C07277=1066.009,101.637,426.334,172.572,27.825,155.091
C07278=1066.003,101.388,426.354,172.570,27.822,155.091
C07279=1065.997,101.139,426.372,172.568,27.819,155.090
C07280=1065.992,100.890,426.391,172.567,27.816,155.090
C07281=1065.985,100.641,426.410,172.565,27.813,155.090
C07282=1065.979,100.391,426.429,172.564,27.811,155.089
C07283=1065.973,100.142,426.448,172.562,27.808,155.089
C07284=1065.967,99.893,426.467,172.561,27.806,155.088
C07285=1065.962,99.645,426.485,172.559,27.803,155.088
C07286=1065.956,99.394,426.504,172.558,27.800,155.088
C07287=1065.950,99.145,426.522,172.556,27.797,155.087
C07288=1065.944,98.896,426.542,172.555,27.794,155.087
C07289=1065.938,98.647,426.560,172.553,27.792,155.086
C07290=1065.933,98.398,426.579,172.551,27.789,155.086
C07291=1065.926,98.149,426.598,172.550,27.787,155.086
C07292=1065.921,97.899,426.616,172.548,27.784,155.085
C07293=1065.914,97.650,426.635,172.547,27.781,155.085
C07294=1065.909,97.400,426.654,172.545,27.778,155.085
C07295=1065.903,97.152,426.673,172.544,27.775,155.084
C07296=1065.897,96.902,426.692,172.542,27.773,155.084
C07297=1065.891,96.653,426.710,172.541,27.770,155.083
C07298=1065.885,96.404,426.728,172.539,27.767,155.083
C07299=1065.879,96.155,426.747,172.538,27.765,155.083
C07300=1065.873,95.906,426.766,172.536,27.762,155.082
C07301=1065.868,95.656,426.784,172.535,27.759,155.082
C07302=1065.861,95.407,426.803,172.533,27.756,155.081
C07303=1065.856,95.158,426.822,172.531,27.754,155.081
C07304=1065.849,94.874,426.843,172.530,27.751,155.081
C07305=1065.843,94.591,426.864,172.529,27.748,155.080
C07306=1065.836,94.307,426.885,172.526,27.745,155.080
C07307=1065.829,94.023,426.906,172.525,27.741,155.079
C07308=1065.823,93.775,426.925,172.523,27.738,155.079
C07309=1065.817,93.525,426.943,172.522,27.736,155.078
C07310=1065.812,93.275,426.962,172.520,27.733,155.078
C07311=1065.806,93.027,426.981,172.519,27.730,155.078
C07312=1065.800,92.777,426.999,172.517,27.728,155.077
C07313=1065.794,92.528,427.018,172.515,27.725,155.077
C07314=1065.788,92.279,427.036,172.514,27.722,155.077
C07315=1065.783,92.029,427.055,172.512,27.719,155.076
C07316=1065.776,91.780,427.073,172.511,27.717,155.076
C07317=1065.772,91.531,427.091,172.510,27.714,155.075
C07318=1065.765,91.282,427.110,172.509,27.711,155.075
C07319=1065.759,91.033,427.129,172.507,27.708,155.075
C07320=1065.754,90.783,427.147,172.506,27.706,155.074
C07321=1065.748,90.534,427.166,172.504,27.703,155.074
C07322=1065.741,90.284,427.184,172.503,27.700,155.073
C07323=1065.736,90.036,427.202,172.501,27.697,155.073
C07324=1065.730,89.786,427.220,172.499,27.695,155.073
C07325=1065.724,89.537,427.239,172.498,27.692,155.072
C07326=1065.717,89.288,427.258,172.496,27.689,155.072
C07327=1065.712,89.039,427.275,172.495,27.687,155.071
C07328=1065.705,88.790,427.294,172.493,27.684,155.071
C07329=1065.700,88.540,427.312,172.492,27.681,155.071
C07330=1065.694,88.291,427.331,172.490,27.679,155.070
C07331=1065.688,88.041,427.349,172.489,27.676,155.070
C07332=1065.682,87.792,427.367,172.487,27.673,155.070
C07333=1065.676,87.543,427.385,172.486,27.670,155.069
C07334=1065.670,87.293,427.403,172.484,27.668,155.069
C07335=1065.664,87.044,427.422,172.483,27.665,155.068
C07336=1065.659,86.795,427.440,172.481,27.663,155.068
C07337=1065.652,86.546,427.458,172.480,27.660,155.068
C07338=1065.647,86.297,427.476,172.478,27.657,155.067
C07339=1065.640,86.048,427.494,172.476,27.654,155.067
C07340=1065.634,85.798,427.512,172.476,27.652,155.066
C07341=1065.629,85.549,427.530,172.474,27.649,155.066
C07342=1065.623,85.299,427.549,172.473,27.646,155.066
C07343=1065.617,85.050,427.567,172.471,27.643,155.065
C07344=1065.611,84.801,427.585,172.470,27.641,155.065
C07345=1065.605,84.552,427.603,172.468,27.638,155.065
C07346=1065.600,84.303,427.621,172.467,27.635,155.064
C07347=1065.593,84.053,427.640,172.465,27.633,155.064
C07348=1065.588,83.804,427.657,172.464,27.630,155.063
C07349=1065.582,83.554,427.676,172.462,27.627,155.063
C07350=1065.576,83.305,427.694,172.461,27.624,155.063
C07351=1065.570,83.056,427.712,172.459,27.621,155.062
C07352=1065.564,82.806,427.730,172.458,27.619,155.062
C07353=1065.558,82.558,427.748,172.456,27.616,155.062
C07354=1065.552,82.308,427.766,172.454,27.614,155.061
C07355=1065.547,82.059,427.784,172.453,27.611,155.061
C07356=1065.541,81.809,427.801,172.451,27.608,155.060
C07357=1065.535,81.561,427.820,172.451,27.605,155.060
C07358=1065.529,81.311,427.838,172.449,27.603,155.059
C07359=1065.523,81.061,427.856,172.448,27.600,155.059
C07360=1065.517,80.813,427.875,172.446,27.597,155.059
C07361=1065.511,80.563,427.892,172.445,27.594,155.058
C07362=1065.506,80.314,427.910,172.443,27.591,155.058
C07363=1065.500,80.064,427.928,172.442,27.589,155.058
C07364=1065.494,79.815,427.946,172.440,27.586,155.057
C07365=1065.488,79.566,427.964,172.439,27.583,155.057
C07366=1065.482,79.317,427.982,172.437,27.581,155.056
C07367=1065.476,79.067,428.000,172.436,27.578,155.056
C07368=1065.470,78.784,428.020,172.434,27.575,155.056
C07369=1065.464,78.500,428.040,172.433,27.572,155.055
C07370=1065.456,78.217,428.060,172.431,27.568,155.055
C07371=1065.449,77.933,428.081,172.429,27.565,155.054
C07372=1065.444,77.684,428.099,172.427,27.563,155.054
C07373=1065.438,77.435,428.117,172.427,27.560,155.053
C07374=1065.432,77.186,428.134,172.425,27.557,155.053
C07375=1065.426,76.936,428.152,172.424,27.555,155.053
C07376=1065.420,76.687,428.169,172.422,27.552,155.052
C07377=1065.414,76.437,428.187,172.421,27.549,155.052
C07378=1065.408,76.189,428.205,172.419,27.547,155.052
C07379=1065.402,75.939,428.223,172.418,27.544,155.051
C07380=1065.396,75.690,428.241,172.416,27.541,155.051
C07381=1065.390,75.440,428.259,172.415,27.539,155.050
C07382=1065.385,75.191,428.276,172.413,27.536,155.050
C07383=1065.379,74.942,428.294,172.412,27.533,155.050
C07384=1065.372,74.693,428.311,172.410,27.530,155.049
C07385=1065.366,74.443,428.329,172.409,27.527,155.049
C07386=1065.361,74.194,428.347,172.407,27.525,155.048
C07387=1065.355,73.944,428.365,172.406,27.522,155.048
C07388=1065.349,73.695,428.382,172.405,27.520,155.048
C07389=1065.343,73.446,428.400,172.403,27.517,155.047
C07390=1065.337,73.197,428.417,172.402,27.514,155.047
C07391=1065.331,72.948,428.435,172.400,27.511,155.047
C07392=1065.325,72.698,428.453,172.399,27.509,155.046
C07393=1065.320,72.449,428.470,172.397,27.506,155.046
C07394=1065.313,72.199,428.488,172.396,27.503,155.045
C07395=1065.308,71.950,428.506,172.394,27.500,155.045
C07396=1065.301,71.701,428.523,172.393,27.498,155.045
C07397=1065.296,71.452,428.541,172.391,27.495,155.044
C07398=1065.290,71.203,428.558,172.390,27.492,155.044
C07399=1065.284,70.953,428.576,172.388,27.489,155.043
C07400=1065.279,70.703,428.593,172.388,27.487,155.043
C07401=1065.272,70.454,428.610,172.386,27.484,155.043
C07402=1065.266,70.205,428.628,172.385,27.481,155.042
C07403=1065.261,69.956,428.646,172.383,27.479,155.042
C07404=1065.255,69.706,428.664,172.382,27.476,155.042
C07405=1065.248,69.457,428.681,172.380,27.473,155.041
C07406=1065.242,69.208,428.698,172.379,27.471,155.041
C07407=1065.237,68.959,428.716,172.377,27.468,155.040
C07408=1065.230,68.708,428.733,172.376,27.465,155.040
C07409=1065.225,68.459,428.750,172.374,27.463,155.040
C07410=1065.219,68.210,428.768,172.372,27.460,155.039
C07411=1065.212,67.961,428.785,172.371,27.457,155.039
C07412=1065.207,67.712,428.803,172.369,27.454,155.039
C07413=1065.202,67.462,428.820,172.369,27.452,155.038
C07414=1065.195,67.213,428.837,172.367,27.449,155.038
C07415=1065.189,66.964,428.854,172.366,27.447,155.037
C07416=1065.183,66.714,428.872,172.364,27.444,155.037
C07417=1065.177,66.465,428.889,172.363,27.441,155.037
C07418=1065.172,66.216,428.906,172.361,27.438,155.036
C07419=1065.165,65.966,428.924,172.360,27.435,155.036
C07420=1065.159,65.717,428.941,172.358,27.433,155.035
C07421=1065.154,65.468,428.959,172.357,27.430,155.035
C07422=1065.147,65.218,428.975,172.355,27.428,155.035
C07423=1065.142,64.969,428.993,172.354,27.425,155.034
C07424=1065.136,64.720,429.010,172.352,27.422,155.034
C07425=1065.130,64.470,429.027,172.352,27.419,155.034
C07426=1065.124,64.221,429.045,172.350,27.417,155.033
C07427=1065.117,63.972,429.062,172.349,27.414,155.033
C07428=1065.111,63.722,429.078,172.347,27.411,155.032
C07429=1065.106,63.473,429.096,172.346,27.409,155.032
C07430=1065.099,63.224,429.113,172.344,27.406,155.032
C07431=1065.094,62.974,429.130,172.342,27.404,155.031
C07432=1065.087,62.690,429.149,172.341,27.401,155.031
C07433=1065.080,62.407,429.169,172.340,27.397,155.030
C07434=1065.073,62.123,429.188,172.337,27.394,155.030
C07435=1065.066,61.839,429.208,172.336,27.391,155.030
C07436=1065.060,61.590,429.225,172.334,27.389,155.029
C07437=1065.053,61.341,429.242,172.333,27.386,155.029
C07438=1065.047,61.091,429.259,172.332,27.384,155.029
C07439=1065.041,60.843,429.276,172.331,27.381,155.028
C07440=1065.035,60.592,429.292,172.329,27.378,155.028
C07441=1065.029,60.343,429.310,172.327,27.376,155.028
C07442=1065.023,60.095,429.327,172.326,27.373,155.027
C07443=1065.017,59.844,429.344,172.324,27.370,155.027
C07444=1065.011,59.596,429.361,172.323,27.368,155.026
C07445=1065.005,59.346,429.377,172.321,27.365,155.026
C07446=1064.999,59.097,429.395,172.320,27.362,155.026
C07447=1064.993,58.847,429.412,172.318,27.360,155.025
C07448=1064.987,58.598,429.429,172.317,27.357,155.025
C07449=1064.981,58.349,429.445,172.316,27.355,155.025
C07450=1064.974,58.099,429.463,172.315,27.352,155.024
C07451=1064.969,57.850,429.479,172.313,27.349,155.024
C07452=1064.963,57.601,429.497,172.312,27.346,155.023
C07453=1064.957,57.352,429.513,172.310,27.344,155.023
C07454=1064.950,57.102,429.530,172.309,27.341,155.023
C07455=1064.945,56.853,429.547,172.307,27.338,155.022
C07456=1064.939,56.603,429.563,172.306,27.336,155.022
C07457=1064.932,56.354,429.581,172.304,27.333,155.022
C07458=1064.927,56.104,429.597,172.303,27.331,155.021
C07459=1064.921,55.855,429.614,172.301,27.328,155.021
C07460=1064.915,55.606,429.631,172.300,27.325,155.020
C07461=1064.909,55.357,429.648,172.299,27.322,155.020
C07462=1064.903,55.107,429.665,172.298,27.320,155.020
C07463=1064.897,54.858,429.681,172.296,27.317,155.019
C07464=1064.891,54.609,429.699,172.295,27.314,155.019
C07465=1064.885,54.359,429.715,172.293,27.312,155.019
C07466=1064.879,54.109,429.732,172.292,27.309,155.018
C07467=1064.872,53.860,429.749,172.290,27.307,155.018
C07468=1064.867,53.611,429.765,172.288,27.304,155.017
C07469=1064.861,53.361,429.782,172.287,27.301,155.017
C07470=1064.855,53.113,429.799,172.286,27.298,155.017
C07471=1064.849,52.862,429.816,172.285,27.296,155.016
C07472=1064.843,52.613,429.832,172.283,27.293,155.016
C07473=1064.837,52.364,429.849,172.282,27.290,155.016
C07474=1064.831,52.115,429.865,172.280,27.288,155.015
C07475=1064.826,51.865,429.882,172.279,27.285,155.015
C07476=1064.820,51.617,429.899,172.277,27.282,155.015
C07477=1064.813,51.366,429.916,172.276,27.280,155.014
C07478=1064.808,51.117,429.933,172.274,27.277,155.014
C07479=1064.802,50.867,429.949,172.273,27.274,155.013
C07480=1064.796,50.619,429.966,172.271,27.271,155.013
C07481=1064.790,50.369,429.982,172.270,27.269,155.013
C07482=1064.784,50.120,429.999,172.269,27.266,155.012
C07483=1064.779,49.870,430.015,172.268,27.264,155.012
C07484=1064.772,49.621,430.033,172.266,27.261,155.011
C07485=1064.766,49.372,430.049,172.265,27.258,155.011
C07486=1064.760,49.122,430.066,172.263,27.256,155.011
C07487=1064.755,48.873,430.082,172.262,27.253,155.010
C07488=1064.749,48.623,430.098,172.260,27.250,155.010
C07489=1064.742,48.375,430.115,172.259,27.247,155.010
C07490=1064.737,48.125,430.132,172.257,27.244,155.009
C07491=1064.731,47.875,430.148,172.256,27.241,155.009
C07492=1064.725,47.626,430.165,172.255,27.239,155.008
C07493=1064.719,47.377,430.181,172.254,27.237,155.008
C07494=1064.713,47.126,430.198,172.252,27.234,155.008
C07495=1064.707,46.878,430.215,172.251,27.231,155.007
C07496=1064.701,46.594,430.234,172.249,27.228,155.007
C07497=1064.694,46.309,430.252,172.248,27.225,155.006
C07498=1064.687,46.026,430.272,172.245,27.222,155.006
C07499=1064.680,45.742,430.290,172.244,27.219,155.006
C07500=1064.675,45.492,430.306,172.243,27.216,155.005
C07501=1064.669,45.243,430.323,172.241,27.213,155.005
C07502=1064.663,44.994,430.339,172.240,27.210,155.004
C07503=1064.657,44.744,430.355,172.239,27.208,155.004
C07504=1064.651,44.495,430.371,172.237,27.205,155.004
C07505=1064.646,44.245,430.388,172.236,27.203,155.003
C07506=1064.640,43.996,430.405,172.235,27.200,155.003
C07507=1064.634,43.746,430.421,172.233,27.197,155.003
C07508=1064.628,43.497,430.437,172.232,27.194,155.002
C07509=1064.622,43.248,430.453,172.230,27.192,155.002
C07510=1064.616,42.998,430.470,172.228,27.189,155.002
C07511=1064.610,42.749,430.486,172.227,27.186,155.001
C07512=1064.604,42.500,430.502,172.226,27.183,155.001
C07513=1064.598,42.250,430.518,172.225,27.181,155.000
C07514=1064.592,42.001,430.535,172.223,27.179,155.000
C07515=1064.586,41.752,430.551,172.222,27.176,155.000
C07516=1064.580,41.502,430.567,172.220,27.173,154.999
C07517=1064.574,41.253,430.583,172.219,27.171,154.999
C07518=1064.569,41.004,430.600,172.217,27.168,154.999
C07519=1064.563,40.754,430.616,172.216,27.165,154.998
C07520=1064.557,40.505,430.632,172.214,27.163,154.998
C07521=1064.551,40.256,430.648,172.213,27.160,154.998
C07522=1064.545,40.006,430.665,172.211,27.157,154.997
C07523=1064.539,39.757,430.681,172.211,27.154,154.997
C07524=1064.533,39.508,430.697,172.209,27.152,154.996
C07525=1064.527,39.258,430.713,172.208,27.149,154.996
C07526=1064.521,39.008,430.729,172.206,27.146,154.996
C07527=1064.515,38.759,430.745,172.205,27.144,154.995
C07528=1064.509,38.510,430.762,172.203,27.141,154.995
C07529=1064.503,38.260,430.778,172.202,27.139,154.995
C07530=1064.497,38.011,430.794,172.200,27.136,154.994
C07531=1064.491,37.761,430.810,172.199,27.133,154.994
C07532=1064.485,37.512,430.826,172.197,27.131,154.993
C07533=1064.479,37.262,430.841,172.197,27.128,154.993
C07534=1064.473,37.013,430.858,172.195,27.126,154.993
C07535=1064.467,36.764,430.874,172.194,27.123,154.992
C07536=1064.461,36.514,430.890,172.192,27.120,154.992
C07537=1064.455,36.265,430.906,172.191,27.118,154.992
C07538=1064.449,36.015,430.921,172.189,27.115,154.991
C07539=1064.443,35.766,430.938,172.188,27.112,154.991
C07540=1064.437,35.517,430.954,172.186,27.110,154.991
C07541=1064.430,35.268,430.970,172.185,27.107,154.990
C07542=1064.425,35.018,430.985,172.183,27.105,154.990
C07543=1064.419,34.768,431.001,172.182,27.102,154.990
C07544=1064.413,34.519,431.018,172.181,27.099,154.989
C07545=1064.406,34.270,431.033,172.180,27.097,154.989
C07546=1064.400,34.020,431.049,172.178,27.094,154.989
C07547=1064.395,33.771,431.065,172.177,27.091,154.988
C07548=1064.389,33.521,431.081,172.175,27.089,154.988
C07549=1064.382,33.272,431.096,172.174,27.086,154.987
C07550=1064.376,33.022,431.113,172.172,27.083,154.987
C07551=1064.370,32.773,431.129,172.171,27.081,154.987
C07552=1064.365,32.523,431.144,172.169,27.078,154.986
C07553=1064.358,32.274,431.160,172.168,27.075,154.986
C07554=1064.352,32.025,431.176,172.166,27.073,154.986
C07555=1064.346,31.775,431.192,172.166,27.071,154.985
C07556=1064.340,31.525,431.208,172.164,27.068,154.985
C07557=1064.334,31.277,431.223,172.163,27.065,154.985
C07558=1064.329,31.027,431.239,172.161,27.063,154.984
C07559=1064.323,30.778,431.255,172.160,27.060,154.984
C07560=1064.315,30.494,431.273,172.158,27.057,154.983
C07561=1064.309,30.209,431.291,172.157,27.054,154.983
C07562=1064.302,29.925,431.309,172.154,27.051,154.983
C07563=1064.295,29.642,431.327,172.153,27.048,154.982
C07564=1064.290,29.392,431.342,172.151,27.045,154.982
C07565=1064.283,29.143,431.358,172.150,27.042,154.982
C07566=1064.277,28.894,431.374,172.149,27.040,154.981
C07567=1064.271,28.644,431.390,172.148,27.038,154.981
C07568=1064.265,28.395,431.405,172.146,27.035,154.981
C07569=1064.259,28.145,431.421,172.145,27.032,154.980
C07570=1064.254,27.896,431.437,172.143,27.030,154.980
C07571=1064.247,27.646,431.452,172.142,27.027,154.979
C07572=1064.241,27.397,431.468,172.140,27.025,154.979
C07573=1064.235,27.147,431.483,172.139,27.022,154.979
C07574=1064.229,26.898,431.499,172.137,27.019,154.978
C07575=1064.223,26.648,431.514,172.136,27.017,154.978
C07576=1064.217,26.399,431.531,172.134,27.014,154.978
C07577=1064.211,26.149,431.546,172.134,27.012,154.977
C07578=1064.205,25.901,431.561,172.132,27.009,154.977
C07579=1064.199,25.651,431.577,172.131,27.007,154.977
C07580=1064.193,25.401,431.592,172.129,27.004,154.976
C07581=1064.187,25.152,431.608,172.128,27.001,154.976
C07582=1064.181,24.902,431.623,172.126,26.999,154.976
C07583=1064.175,24.653,431.639,172.125,26.996,154.975
C07584=1064.168,24.403,431.654,172.123,26.993,154.975
C07585=1064.163,24.154,431.669,172.122,26.991,154.975
C07586=1064.157,23.905,431.685,172.120,26.988,154.974
C07587=1064.151,23.655,431.701,172.119,26.986,154.974
C07588=1064.144,23.406,431.716,172.118,26.983,154.974
C07589=1064.139,23.156,431.732,172.117,26.981,154.973
C07590=1064.133,22.907,431.746,172.115,26.978,154.973
C07591=1064.127,22.657,431.763,172.114,26.976,154.973
C07592=1064.121,22.408,431.778,172.112,26.973,154.972
C07593=1064.115,22.158,431.793,172.111,26.970,154.972
C07594=1064.108,21.909,431.809,172.109,26.968,154.972
C07595=1064.103,21.659,431.824,172.108,26.965,154.971
C07596=1064.097,21.410,431.839,172.106,26.963,154.971
C07597=1064.090,21.161,431.855,172.105,26.960,154.971
C07598=1064.084,20.911,431.870,172.103,26.957,154.970
C07599=1064.078,20.661,431.885,172.102,26.955,154.970
C07600=1064.073,20.413,431.901,172.101,26.952,154.969
C07601=1064.066,20.163,431.916,172.099,26.950,154.969
C07602=1064.061,19.913,431.931,172.098,26.947,154.969
C07603=1064.054,19.663,431.946,172.096,26.945,154.969
C07604=1064.048,19.415,431.962,172.095,26.942,154.968
C07605=1064.043,19.165,431.977,172.093,26.940,154.968
C07606=1064.036,18.915,431.992,172.092,26.937,154.967
C07607=1064.030,18.666,432.007,172.090,26.935,154.967
C07608=1064.024,18.416,432.023,172.089,26.932,154.967
C07609=1064.018,18.167,432.038,172.087,26.930,154.967
C07610=1064.012,17.917,432.054,172.086,26.927,154.966
C07611=1064.006,17.668,432.068,172.085,26.925,154.966
C07612=1064.000,17.419,432.083,172.084,26.922,154.965
C07613=1063.995,17.169,432.099,172.082,26.920,154.965
C07614=1063.988,16.920,432.114,172.081,26.917,154.965
C07615=1063.982,16.670,432.129,172.079,26.914,154.964
C07616=1063.976,16.421,432.144,172.078,26.912,154.964
C07617=1063.970,16.171,432.159,172.076,26.909,154.964
C07618=1063.964,15.921,432.174,172.075,26.906,154.963
C07619=1063.958,15.672,432.190,172.073,26.904,154.963
C07620=1063.952,15.423,432.205,172.072,26.901,154.963
C07621=1063.946,15.174,432.220,172.070,26.899,154.963
C07622=1063.939,14.924,432.235,172.069,26.896,154.962
C07623=1063.934,14.675,432.250,172.067,26.894,154.962
C07624=1063.927,14.392,432.267,172.066,26.891,154.961
C07625=1063.920,14.110,432.284,172.064,26.888,154.961
C07626=1063.913,13.826,432.302,172.063,26.885,154.961
C07627=1063.907,13.544,432.318,172.061,26.882,154.960
C07628=1063.900,13.295,432.333,172.060,26.880,154.960
C07629=1063.894,13.045,432.348,172.058,26.877,154.960
C07630=1063.887,12.795,432.363,172.057,26.875,154.959
C07631=1063.882,12.546,432.378,172.055,26.873,154.959
C07632=1063.875,12.297,432.393,172.054,26.870,154.959
C07633=1063.869,12.047,432.408,172.052,26.868,154.958
C07634=1063.863,11.798,432.422,172.051,26.865,154.958
C07635=1063.857,11.548,432.438,172.049,26.862,154.958
C07636=1063.851,11.298,432.453,172.048,26.860,154.957
C07637=1063.845,11.049,432.468,172.047,26.858,154.957
C07638=1063.839,10.800,432.482,172.046,26.855,154.957
C07639=1063.833,10.550,432.497,172.044,26.853,154.957
C07640=1063.826,10.301,432.512,172.043,26.850,154.956
C07641=1063.820,10.052,432.527,172.041,26.848,154.956
C07642=1063.814,9.802,432.542,172.040,26.846,154.956
C07643=1063.808,9.552,432.556,172.038,26.843,154.955
C07644=1063.802,9.303,432.570,172.037,26.840,154.955
C07645=1063.796,9.053,432.585,172.035,26.838,154.955
C07646=1063.789,8.803,432.600,172.034,26.835,154.954
C07647=1063.784,8.554,432.615,172.032,26.833,154.954
C07648=1063.778,8.304,432.630,172.031,26.830,154.954
C07649=1063.772,8.055,432.645,172.029,26.828,154.953
C07650=1063.766,7.806,432.660,172.028,26.826,154.953
C07651=1063.759,7.556,432.675,172.026,26.823,154.953
C07652=1063.754,7.307,432.689,172.025,26.821,154.952
C07653=1063.748,7.057,432.704,172.024,26.818,154.952
C07654=1063.741,6.807,432.719,172.022,26.816,154.952
C07655=1063.735,6.558,432.733,172.021,26.813,154.951
C07656=1063.729,6.309,432.748,172.019,26.810,154.951
C07657=1063.723,6.060,432.763,172.018,26.808,154.951
C07658=1063.717,5.810,432.778,172.016,26.806,154.951
C07659=1063.711,5.560,432.792,172.015,26.803,154.950
C07660=1063.705,5.311,432.807,172.013,26.801,154.950
C07661=1063.699,5.061,432.821,172.012,26.798,154.950
C07662=1063.693,4.812,432.836,172.010,26.795,154.949
C07663=1063.686,4.563,432.851,172.009,26.793,154.949
C07664=1063.681,4.313,432.865,172.007,26.790,154.949
C07665=1063.675,4.063,432.880,172.006,26.788,154.948
C07666=1063.668,3.814,432.895,172.005,26.786,154.948
C07667=1063.662,3.565,432.909,172.004,26.783,154.948
C07668=1063.656,3.314,432.924,172.002,26.781,154.947
C07669=1063.650,3.066,432.938,172.001,26.779,154.947
C07670=1063.644,2.816,432.953,171.999,26.776,154.947
C07671=1063.639,2.566,432.967,171.998,26.773,154.946
C07672=1063.632,2.317,432.982,171.996,26.771,154.946
C07673=1063.626,2.068,432.996,171.995,26.768,154.946
C07674=1063.620,1.818,433.011,171.993,26.766,154.945
C07675=1063.615,1.568,433.025,171.992,26.763,154.945
C07676=1063.608,1.319,433.040,171.990,26.761,154.945
C07677=1063.602,1.070,433.055,171.989,26.759,154.945
C07678=1063.596,0.820,433.069,171.987,26.756,154.944
C07679=1063.591,0.571,433.084,171.986,26.753,154.944
C07680=1063.584,0.321,433.099,171.984,26.751,154.944
C07681=1063.579,0.071,433.112,171.983,26.748,154.943
C07682=1063.572,-0.178,433.127,171.982,26.746,154.943
C07683=1063.567,-0.428,433.141,171.981,26.744,154.943
C07684=1063.560,-0.678,433.156,171.979,26.741,154.942
C07685=1063.555,-0.926,433.171,171.978,26.739,154.942
C07686=1063.549,-1.177,433.185,171.976,26.736,154.942
C07687=1063.543,-1.426,433.200,171.975,26.734,154.941
C07688=1063.537,-1.707,433.216,171.973,26.731,154.941
C07689=1063.529,-1.988,433.232,171.971,26.728,154.941
C07690=1063.523,-2.267,433.248,171.969,26.725,154.940
C07691=1063.516,-2.548,433.264,171.968,26.722,154.940
C07692=1063.510,-2.797,433.279,171.966,26.720,154.940
C07693=1063.504,-3.048,433.293,171.965,26.718,154.939
C07694=1063.498,-3.297,433.308,171.963,26.715,154.939
C07695=1063.492,-3.547,433.322,171.962,26.713,154.939
C07696=1063.486,-3.796,433.336,171.960,26.710,154.938
C07697=1063.480,-4.046,433.350,171.959,26.708,154.938
C07698=1063.474,-4.295,433.365,171.957,26.706,154.938
C07699=1063.468,-4.545,433.379,171.957,26.703,154.937
C07700=1063.462,-4.794,433.393,171.955,26.701,154.937
C07701=1063.455,-5.044,433.407,171.954,26.699,154.937
C07702=1063.449,-5.293,433.422,171.952,26.696,154.937
C07703=1063.443,-5.543,433.436,171.950,26.694,154.936
C07704=1063.437,-5.793,433.449,171.949,26.692,154.936
C07705=1063.431,-6.042,433.464,171.947,26.689,154.936
C07706=1063.425,-6.292,433.478,171.946,26.686,154.935
C07707=1063.419,-6.540,433.492,171.944,26.684,154.935
C07708=1063.413,-6.791,433.506,171.943,26.682,154.935
C07709=1063.407,-7.040,433.521,171.941,26.680,154.935
C07710=1063.400,-7.290,433.534,171.940,26.677,154.934
C07711=1063.394,-7.539,433.548,171.938,26.674,154.934
C07712=1063.388,-7.789,433.563,171.937,26.672,154.934
C07713=1063.382,-8.038,433.576,171.935,26.670,154.933
C07714=1063.376,-8.287,433.591,171.934,26.668,154.933
C07715=1063.370,-8.537,433.605,171.932,26.665,154.933
C07716=1063.364,-8.787,433.619,171.931,26.663,154.933
C07717=1063.357,-9.036,433.633,171.929,26.660,154.932
C07718=1063.352,-9.286,433.647,171.928,26.658,154.932
C07719=1063.346,-9.535,433.661,171.926,26.655,154.932
C07720=1063.339,-9.785,433.676,171.925,26.653,154.931
C07721=1063.334,-10.034,433.689,171.924,26.651,154.931
C07722=1063.327,-10.284,433.703,171.922,26.649,154.931
C07723=1063.322,-10.534,433.717,171.921,26.647,154.931
C07724=1063.316,-10.783,433.732,171.919,26.644,154.930
C07725=1063.309,-11.033,433.745,171.918,26.641,154.930
C07726=1063.304,-11.282,433.759,171.916,26.639,154.930
C07727=1063.297,-11.531,433.773,171.915,26.637,154.929
C07728=1063.291,-11.781,433.787,171.913,26.634,154.929
C07729=1063.285,-12.031,433.801,171.912,26.632,154.929
C07730=1063.279,-12.280,433.814,171.910,26.630,154.929
C07731=1063.273,-12.530,433.829,171.909,26.628,154.928
C07732=1063.267,-12.779,433.843,171.907,26.625,154.928
C07733=1063.261,-13.029,433.856,171.906,26.622,154.928
C07734=1063.255,-13.279,433.871,171.904,26.620,154.927
C07735=1063.249,-13.528,433.884,171.903,26.618,154.927
C07736=1063.243,-13.777,433.899,171.901,26.615,154.927
C07737=1063.237,-14.027,433.913,171.900,26.613,154.927
C07738=1063.231,-14.277,433.926,171.898,26.611,154.926
C07739=1063.225,-14.526,433.940,171.896,26.609,154.926
C07740=1063.219,-14.776,433.954,171.895,26.606,154.926
C07741=1063.213,-15.025,433.968,171.894,26.603,154.925
C07742=1063.207,-15.274,433.981,171.892,26.601,154.925
C07743=1063.200,-15.525,433.996,171.890,26.599,154.925
C07744=1063.194,-15.774,434.009,171.889,26.596,154.925
C07745=1063.189,-16.024,434.023,171.887,26.594,154.924
C07746=1063.182,-16.273,434.036,171.886,26.592,154.924
C07747=1063.176,-16.523,434.050,171.884,26.590,154.924
C07748=1063.170,-16.772,434.064,171.883,26.587,154.924
C07749=1063.164,-17.022,434.077,171.882,26.585,154.923
C07750=1063.158,-17.271,434.092,171.881,26.583,154.923
C07751=1063.151,-17.521,434.105,171.879,26.581,154.923
C07752=1063.145,-17.799,434.120,171.877,26.578,154.923
C07753=1063.138,-18.079,434.135,171.875,26.576,154.922
C07754=1063.131,-18.358,434.150,171.874,26.573,154.922
C07755=1063.124,-18.637,434.165,171.872,26.571,154.922
C07756=1063.118,-18.887,434.179,171.871,26.568,154.921
C07757=1063.112,-19.136,434.193,171.869,26.566,154.921
C07758=1063.106,-19.386,434.207,171.868,26.564,154.921
C07759=1063.100,-19.635,434.220,171.866,26.561,154.921
C07760=1063.093,-19.885,434.233,171.864,26.559,154.920
C07761=1063.088,-20.135,434.247,171.863,26.557,154.920
C07762=1063.082,-20.384,434.261,171.861,26.554,154.920
C07763=1063.075,-20.633,434.274,171.860,26.553,154.920
C07764=1063.069,-20.884,434.288,171.858,26.550,154.919
C07765=1063.063,-21.133,434.301,171.857,26.548,154.919
C07766=1063.058,-21.382,434.315,171.855,26.546,154.919
C07767=1063.051,-21.632,434.328,171.854,26.543,154.919
C07768=1063.045,-21.882,434.342,171.852,26.541,154.918
C07769=1063.039,-22.131,434.356,171.851,26.539,154.918
C07770=1063.033,-22.380,434.369,171.849,26.537,154.918
C07771=1063.027,-22.630,434.382,171.848,26.534,154.917
C07772=1063.021,-22.879,434.396,171.846,26.532,154.917
C07773=1063.014,-23.129,434.410,171.844,26.530,154.917
C07774=1063.008,-23.379,434.423,171.843,26.527,154.917
C07775=1063.003,-23.629,434.436,171.841,26.525,154.916
C07776=1062.997,-23.878,434.450,171.840,26.523,154.916
C07777=1062.991,-24.127,434.463,171.838,26.520,154.916
C07778=1062.985,-24.377,434.477,171.837,26.518,154.916
C07779=1062.978,-24.627,434.490,171.835,26.516,154.915
C07780=1062.972,-24.876,434.504,171.834,26.514,154.915
C07781=1062.966,-25.125,434.517,171.832,26.512,154.915
C07782=1062.961,-25.376,434.530,171.831,26.509,154.915
C07783=1062.954,-25.625,434.543,171.829,26.507,154.914
C07784=1062.948,-25.874,434.557,171.827,26.505,154.914
C07785=1062.942,-26.124,434.571,171.826,26.502,154.914
C07786=1062.936,-26.374,434.584,171.824,26.500,154.914
C07787=1062.930,-26.623,434.597,171.823,26.498,154.913
C07788=1062.925,-26.873,434.611,171.821,26.496,154.913
C07789=1062.918,-27.122,434.624,171.820,26.494,154.913
C07790=1062.912,-27.372,434.637,171.818,26.491,154.913
C07791=1062.905,-27.622,434.651,171.817,26.489,154.912
C07792=1062.899,-27.871,434.663,171.815,26.487,154.912
C07793=1062.893,-28.121,434.677,171.814,26.485,154.912
C07794=1062.887,-28.370,434.690,171.812,26.483,154.912
C07795=1062.881,-28.619,434.703,171.810,26.480,154.911
C07796=1062.875,-28.869,434.716,171.809,26.478,154.911
C07797=1062.869,-29.118,434.729,171.807,26.476,154.911
C07798=1062.863,-29.369,434.743,171.806,26.474,154.911
C07799=1062.857,-29.619,434.756,171.804,26.472,154.910
C07800=1062.850,-29.868,434.769,171.803,26.470,154.910
C07801=1062.844,-30.117,434.782,171.801,26.468,154.910
C07802=1062.838,-30.367,434.795,171.800,26.465,154.910
C07803=1062.832,-30.616,434.808,171.798,26.463,154.910
C07804=1062.826,-30.865,434.821,171.796,26.461,154.909
C07805=1062.819,-31.116,434.834,171.795,26.459,154.909
C07806=1062.813,-31.365,434.848,171.793,26.457,154.909
C07807=1062.807,-31.615,434.861,171.792,26.454,154.909
C07808=1062.801,-31.864,434.873,171.790,26.452,154.908
C07809=1062.795,-32.114,434.887,171.789,26.450,154.908
C07810=1062.789,-32.364,434.899,171.787,26.448,154.908
C07811=1062.783,-32.613,434.912,171.786,26.446,154.908
C07812=1062.776,-32.862,434.926,171.784,26.444,154.907
C07813=1062.771,-33.112,434.939,171.782,26.442,154.907
C07814=1062.765,-33.362,434.952,171.781,26.439,154.907
C07815=1062.759,-33.611,434.965,171.779,26.437,154.907
C07816=1062.752,-33.890,434.979,171.778,26.435,154.906
C07817=1062.745,-34.168,434.994,171.776,26.432,154.906
C07818=1062.738,-34.446,435.009,171.775,26.430,154.906
C07819=1062.731,-34.724,435.023,171.773,26.428,154.906
C07820=1062.725,-34.974,435.035,171.772,26.426,154.905
C07821=1062.720,-35.224,435.049,171.770,26.424,154.905
C07822=1062.714,-35.473,435.062,171.769,26.421,154.905
C07823=1062.708,-35.723,435.075,171.767,26.420,154.905
C07824=1062.702,-35.973,435.088,171.765,26.417,154.905
C07825=1062.695,-36.222,435.101,171.763,26.415,154.904
C07826=1062.690,-36.472,435.113,171.761,26.413,154.904
C07827=1062.683,-36.721,435.127,171.760,26.411,154.904
C07828=1062.677,-36.971,435.139,171.758,26.408,154.904
C07829=1062.671,-37.220,435.152,171.757,26.407,154.904
C07830=1062.665,-37.470,435.165,171.755,26.404,154.903
C07831=1062.659,-37.719,435.178,171.754,26.402,154.903
C07832=1062.653,-37.969,435.191,171.752,26.400,154.903
C07833=1062.647,-38.219,435.203,171.750,26.398,154.903
C07834=1062.641,-38.468,435.217,171.749,26.396,154.902
C07835=1062.635,-38.718,435.229,171.747,26.394,154.902
C07836=1062.628,-38.967,435.242,171.746,26.392,154.902
C07837=1062.622,-39.217,435.254,171.744,26.390,154.902
C07838=1062.616,-39.467,435.267,171.743,26.388,154.901
C07839=1062.610,-39.716,435.280,171.741,26.386,154.901
C07840=1062.604,-39.966,435.293,171.739,26.384,154.901
C07841=1062.598,-40.216,435.305,171.738,26.382,154.901
C07842=1062.591,-40.465,435.318,171.736,26.379,154.901
C07843=1062.585,-40.715,435.331,171.735,26.378,154.901
C07844=1062.579,-40.964,435.344,171.733,26.375,154.900
C07845=1062.573,-41.214,435.356,171.731,26.374,154.900
C07846=1062.567,-41.463,435.368,171.730,26.371,154.900
C07847=1062.561,-41.713,435.381,171.728,26.370,154.900
C07848=1062.555,-41.963,435.394,171.727,26.367,154.899
C07849=1062.549,-42.213,435.407,171.725,26.366,154.899
C07850=1062.542,-42.462,435.419,171.724,26.363,154.899
C07851=1062.536,-42.711,435.432,171.722,26.361,154.899
C07852=1062.530,-42.961,435.445,171.720,26.359,154.899
C07853=1062.524,-43.211,435.457,171.719,26.357,154.898
C07854=1062.518,-43.461,435.470,171.717,26.355,154.898
C07855=1062.511,-43.710,435.482,171.716,26.353,154.898
C07856=1062.505,-43.960,435.495,171.714,26.351,154.898
C07857=1062.499,-44.210,435.507,171.713,26.349,154.898
C07858=1062.494,-44.459,435.520,171.711,26.347,154.897
C07859=1062.487,-44.708,435.532,171.709,26.345,154.897
C07860=1062.481,-44.958,435.545,171.708,26.343,154.897
C07861=1062.475,-45.208,435.557,171.706,26.341,154.897
C07862=1062.469,-45.457,435.570,171.705,26.339,154.897
C07863=1062.463,-45.707,435.582,171.703,26.337,154.896
C07864=1062.456,-45.956,435.595,171.701,26.335,154.896
C07865=1062.451,-46.206,435.608,171.700,26.333,154.896
C07866=1062.445,-46.456,435.620,171.698,26.331,154.896
C07867=1062.438,-46.706,435.632,171.697,26.329,154.896
C07868=1062.433,-46.955,435.644,171.695,26.327,154.895
C07869=1062.427,-47.205,435.657,171.694,26.325,154.895
C07870=1062.420,-47.454,435.670,171.692,26.323,154.895
C07871=1062.414,-47.704,435.682,171.690,26.321,154.895
C07872=1062.408,-47.953,435.695,171.689,26.319,154.895
C07873=1062.402,-48.203,435.707,171.687,26.317,154.895
C07874=1062.395,-48.453,435.719,171.686,26.315,154.894
C07875=1062.390,-48.702,435.731,171.684,26.313,154.894
C07876=1062.384,-48.952,435.744,171.682,26.312,154.894
C07877=1062.378,-49.202,435.756,171.681,26.309,154.894
C07878=1062.372,-49.451,435.769,171.679,26.307,154.894
C07879=1062.366,-49.701,435.781,171.678,26.305,154.893
C07880=1062.359,-49.980,435.795,171.675,26.303,154.893
C07881=1062.352,-50.259,435.808,171.674,26.301,154.893
C07882=1062.345,-50.536,435.822,171.672,26.299,154.893
C07883=1062.338,-50.815,435.836,171.671,26.297,154.893
C07884=1062.333,-51.065,435.848,171.669,26.295,154.892
C07885=1062.326,-51.314,435.860,171.666,26.293,154.892
C07886=1062.319,-51.564,435.872,171.665,26.291,154.892
C07887=1062.313,-51.814,435.885,171.663,26.289,154.892
C07888=1062.307,-52.063,435.897,171.662,26.287,154.892
C07889=1062.301,-52.313,435.909,171.660,26.285,154.892
C07890=1062.294,-52.563,435.921,171.658,26.284,154.891
C07891=1062.289,-52.813,435.933,171.657,26.282,154.891
C07892=1062.282,-53.062,435.945,171.655,26.280,154.891
C07893=1062.276,-53.312,435.957,171.653,26.278,154.891
C07894=1062.270,-53.562,435.969,171.652,26.276,154.891
C07895=1062.263,-53.811,435.981,171.650,26.274,154.891
C07896=1062.257,-54.061,435.994,171.649,26.273,154.890
C07897=1062.251,-54.311,436.006,171.647,26.271,154.890
C07898=1062.245,-54.559,436.017,171.645,26.269,154.890
C07899=1062.239,-54.809,436.030,171.644,26.267,154.890
C07900=1062.232,-55.059,436.042,171.642,26.265,154.890
C07901=1062.225,-55.308,436.054,171.641,26.263,154.890
C07902=1062.220,-55.559,436.066,171.639,26.262,154.889
C07903=1062.214,-55.808,436.077,171.637,26.260,154.889
C07904=1062.208,-56.058,436.090,171.636,26.258,154.889
C07905=1062.201,-56.307,436.102,171.634,26.256,154.889
C07906=1062.195,-56.557,436.114,171.632,26.255,154.889
C07907=1062.189,-56.807,436.126,171.631,26.253,154.889
C07908=1062.183,-57.056,436.138,171.629,26.250,154.889
C07909=1062.176,-57.306,436.149,171.628,26.249,154.888
C07910=1062.170,-57.556,436.162,171.626,26.247,154.888
C07911=1062.164,-57.805,436.174,171.624,26.245,154.888
C07912=1062.158,-58.054,436.185,171.622,26.243,154.888
C07913=1062.152,-58.304,436.198,171.620,26.241,154.888
C07914=1062.146,-58.554,436.209,171.619,26.240,154.888
C07915=1062.139,-58.804,436.221,171.617,26.238,154.888
C07916=1062.134,-59.053,436.233,171.615,26.236,154.887
C07917=1062.127,-59.303,436.245,171.614,26.234,154.887
C07918=1062.121,-59.553,436.256,171.612,26.233,154.887
C07919=1062.115,-59.803,436.269,171.610,26.231,154.887
C07920=1062.109,-60.051,436.281,171.609,26.229,154.887
C07921=1062.102,-60.301,436.293,171.607,26.227,154.887
C07922=1062.096,-60.552,436.304,171.606,26.225,154.886
C07923=1062.090,-60.800,436.316,171.604,26.223,154.886
C07924=1062.084,-61.050,436.328,171.602,26.222,154.886
C07925=1062.078,-61.301,436.340,171.601,26.220,154.886
C07926=1062.071,-61.550,436.352,171.599,26.218,154.886
C07927=1062.065,-61.799,436.363,171.597,26.216,154.886
C07928=1062.060,-62.049,436.375,171.596,26.215,154.886
C07929=1062.053,-62.299,436.387,171.594,26.213,154.885
C07930=1062.047,-62.548,436.399,171.593,26.211,154.885
C07931=1062.041,-62.798,436.411,171.591,26.209,154.885
C07932=1062.035,-63.048,436.423,171.589,26.208,154.885
C07933=1062.029,-63.297,436.434,171.588,26.206,154.885
C07934=1062.022,-63.547,436.445,171.586,26.204,154.885
C07935=1062.017,-63.796,436.458,171.584,26.202,154.885
C07936=1062.010,-64.046,436.470,171.582,26.200,154.885
C07937=1062.004,-64.296,436.481,171.580,26.199,154.884
C07938=1061.999,-64.545,436.493,171.579,26.197,154.884
C07939=1061.993,-64.795,436.504,171.577,26.195,154.884
C07940=1061.986,-65.045,436.516,171.575,26.193,154.884
C07941=1061.980,-65.294,436.528,171.574,26.192,154.884
C07942=1061.974,-65.544,436.540,171.572,26.190,154.884
C07943=1061.968,-65.793,436.551,171.570,26.188,154.884
C07944=1061.959,-66.139,436.567,171.568,26.186,154.883
C07945=1061.951,-66.484,436.584,171.566,26.184,154.883
C07946=1061.942,-66.830,436.599,171.564,26.181,154.883
C07947=1061.935,-67.175,436.615,171.561,26.179,154.883
C07948=1061.928,-67.425,436.627,171.560,26.177,154.883
C07949=1061.923,-67.674,436.638,171.558,26.176,154.883
C07950=1061.916,-67.924,436.650,171.557,26.174,154.882
C07951=1061.910,-68.174,436.661,171.555,26.172,154.882
C07952=1061.904,-68.423,436.674,171.553,26.170,154.882
C07953=1061.898,-68.673,436.685,171.552,26.169,154.882
C07954=1061.892,-68.922,436.696,171.550,26.167,154.882
C07955=1061.886,-69.172,436.708,171.547,26.165,154.882
C07956=1061.880,-69.422,436.720,171.546,26.164,154.882
C07957=1061.874,-69.672,436.731,171.544,26.162,154.882
C07958=1061.868,-69.921,436.743,171.542,26.160,154.881
C07959=1061.862,-70.171,436.754,171.541,26.158,154.881
C07960=1061.857,-70.421,436.765,171.539,26.157,154.881
C07961=1061.850,-70.670,436.777,171.538,26.155,154.881
C07962=1061.844,-70.920,436.788,171.536,26.153,154.881
C07963=1061.838,-71.169,436.800,171.534,26.151,154.881
C07964=1061.832,-71.419,436.811,171.533,26.150,154.881
C07965=1061.826,-71.669,436.823,171.531,26.148,154.881
C07966=1061.820,-71.918,436.835,171.529,26.147,154.880
C07967=1061.814,-72.168,436.846,171.528,26.145,154.880
C07968=1061.808,-72.418,436.857,171.526,26.143,154.880
C07969=1061.801,-72.667,436.869,171.524,26.141,154.880
C07970=1061.796,-72.917,436.880,171.523,26.140,154.880
C07971=1061.790,-73.167,436.891,171.521,26.138,154.880
C07972=1061.784,-73.416,436.903,171.519,26.137,154.880
C07973=1061.778,-73.666,436.914,171.518,26.135,154.880
C07974=1061.772,-73.916,436.925,171.516,26.133,154.879
C07975=1061.765,-74.165,436.937,171.514,26.132,154.879
C07976=1061.760,-74.415,436.948,171.512,26.130,154.879
C07977=1061.753,-74.665,436.959,171.510,26.128,154.879
C07978=1061.747,-74.914,436.971,171.509,26.127,154.879
C07979=1061.741,-75.164,436.982,171.507,26.125,154.879
C07980=1061.735,-75.414,436.993,171.505,26.124,154.879
C07981=1061.729,-75.664,437.004,171.504,26.122,154.879
C07982=1061.723,-75.913,437.016,171.502,26.121,154.879
C07983=1061.716,-76.163,437.027,171.500,26.119,154.879
C07984=1061.711,-76.412,437.038,171.499,26.118,154.879
C07985=1061.705,-76.662,437.049,171.497,26.116,154.878
C07986=1061.699,-76.912,437.060,171.495,26.114,154.878
C07987=1061.692,-77.161,437.072,171.494,26.113,154.878
C07988=1061.686,-77.411,437.083,171.492,26.111,154.878
C07989=1061.680,-77.661,437.094,171.490,26.110,154.878
C07990=1061.674,-77.911,437.105,171.489,26.108,154.878
C07991=1061.668,-78.160,437.116,171.487,26.107,154.878
C07992=1061.662,-78.410,437.128,171.485,26.105,154.878
C07993=1061.656,-78.659,437.139,171.484,26.104,154.878
C07994=1061.649,-78.909,437.149,171.481,26.102,154.878
C07995=1061.643,-79.159,437.160,171.479,26.100,154.878
C07996=1061.637,-79.408,437.171,171.478,26.099,154.877
C07997=1061.631,-79.658,437.182,171.476,26.097,154.877
C07998=1061.625,-79.908,437.193,171.474,26.096,154.877
C07999=1061.619,-80.158,437.204,171.473,26.095,154.877
C08000=1061.613,-80.375,437.214,171.471,26.093,154.877
C08001=1061.608,-80.592,437.223,171.470,26.092,154.877
C08002=1061.603,-80.809,437.232,171.468,26.091,154.877
C08003=1061.598,-81.025,437.243,171.467,26.090,154.877
C08004=1061.592,-81.243,437.252,171.465,26.088,154.877
C08005=1061.586,-81.460,437.261,171.463,26.087,154.877
C08006=1061.581,-81.676,437.271,171.462,26.086,154.877
C08007=1061.575,-81.893,437.280,171.461,26.085,154.877
C08008=1061.568,-82.176,437.293,171.459,26.083,154.877
C08009=1061.562,-82.458,437.305,171.456,26.081,154.877
C08010=1061.554,-82.740,437.318,171.455,26.080,154.876
C08011=1061.548,-83.022,437.329,171.453,26.078,154.876
C08012=1061.541,-83.273,437.340,171.450,26.076,154.876
C08013=1061.535,-83.522,437.351,171.449,26.075,154.876
C08014=1061.529,-83.772,437.362,171.447,26.074,154.876
C08015=1061.523,-84.021,437.373,171.445,26.072,154.876
C08016=1061.517,-84.271,437.384,171.444,26.071,154.876
C08017=1061.510,-84.521,437.394,171.442,26.070,154.876
C08018=1061.504,-84.770,437.405,171.440,26.068,154.876
C08019=1061.498,-85.020,437.417,171.439,26.067,154.876
C08020=1061.492,-85.270,437.427,171.437,26.066,154.876
C08021=1061.486,-85.519,437.438,171.435,26.064,154.876
C08022=1061.479,-85.769,437.449,171.433,26.063,154.876
C08023=1061.473,-86.018,437.459,171.432,26.062,154.876
C08024=1061.467,-86.268,437.470,171.430,26.060,154.876
C08025=1061.461,-86.518,437.481,171.428,26.059,154.876
C08026=1061.454,-86.767,437.492,171.427,26.058,154.876
C08027=1061.449,-87.017,437.502,171.425,26.056,154.875
C08028=1061.442,-87.267,437.514,171.423,26.055,154.875
C08029=1061.436,-87.517,437.523,171.421,26.053,154.875
C08030=1061.430,-87.766,437.534,171.419,26.052,154.875
C08031=1061.424,-88.016,437.545,171.417,26.050,154.875
C08032=1061.418,-88.266,437.556,171.415,26.049,154.875
C08033=1061.412,-88.515,437.567,171.414,26.048,154.875
C08034=1061.406,-88.765,437.578,171.412,26.046,154.875
C08035=1061.399,-89.015,437.588,171.410,26.045,154.875
C08036=1061.394,-89.265,437.598,171.409,26.044,154.875
C08037=1061.387,-89.515,437.609,171.407,26.043,154.875
C08038=1061.381,-89.764,437.620,171.405,26.041,154.875
C08039=1061.375,-90.013,437.631,171.403,26.040,154.875
C08040=1061.369,-90.263,437.642,171.402,26.039,154.875
C08041=1061.363,-90.513,437.651,171.400,26.037,154.875
C08042=1061.357,-90.763,437.662,171.398,26.036,154.875
C08043=1061.350,-91.012,437.673,171.397,26.034,154.875
C08044=1061.345,-91.262,437.683,171.395,26.033,154.875
C08045=1061.338,-91.512,437.695,171.392,26.032,154.875
C08046=1061.332,-91.762,437.704,171.390,26.031,154.875
C08047=1061.326,-92.011,437.715,171.389,26.029,154.875
C08048=1061.320,-92.260,437.725,171.387,26.028,154.875
C08049=1061.314,-92.511,437.736,171.385,26.026,154.874
C08050=1061.308,-92.761,437.747,171.384,26.025,154.874
C08051=1061.302,-93.010,437.757,171.382,26.024,154.874
C08052=1061.296,-93.259,437.768,171.380,26.023,154.874
C08053=1061.290,-93.510,437.779,171.379,26.021,154.874
C08054=1061.283,-93.759,437.789,171.377,26.020,154.874
C08055=1061.278,-94.009,437.800,171.375,26.019,154.874
C08056=1061.271,-94.259,437.809,171.373,26.018,154.874
C08057=1061.266,-94.508,437.820,171.372,26.017,154.874
C08058=1061.259,-94.757,437.830,171.370,26.015,154.874
C08059=1061.253,-95.008,437.841,171.368,26.014,154.874
C08060=1061.247,-95.258,437.852,171.366,26.012,154.874
C08061=1061.241,-95.507,437.862,171.365,26.011,154.874
C08062=1061.236,-95.757,437.872,171.362,26.010,154.874
C08063=1061.229,-96.006,437.883,171.360,26.009,154.874
C08064=1061.223,-96.256,437.894,171.359,26.007,154.874
C08065=1061.217,-96.506,437.904,171.357,26.006,154.874
C08066=1061.211,-96.755,437.914,171.355,26.005,154.874
C08067=1061.205,-97.006,437.924,171.353,26.004,154.874
C08068=1061.199,-97.255,437.935,171.352,26.003,154.874
C08069=1061.193,-97.505,437.945,171.350,26.002,154.874
C08070=1061.186,-97.755,437.956,171.348,26.000,154.874
C08071=1061.180,-98.004,437.966,171.346,25.999,154.874
C08072=1061.173,-98.289,437.978,171.345,25.998,154.874
C08073=1061.166,-98.573,437.990,171.342,25.997,154.874
C08074=1061.159,-98.858,438.001,171.340,25.995,154.874
C08075=1061.152,-99.142,438.013,171.339,25.994,154.874
C08076=1061.146,-99.392,438.023,171.336,25.993,154.874
C08077=1061.140,-99.641,438.033,171.334,25.992,154.874
C08078=1061.134,-99.891,438.043,171.332,25.990,154.874
C08079=1061.128,-100.140,438.053,171.331,25.989,154.874
C08080=1061.122,-100.390,438.063,171.329,25.988,154.874
C08081=1061.116,-100.640,438.074,171.327,25.987,154.874
C08082=1061.109,-100.890,438.084,171.325,25.986,154.874
C08083=1061.103,-101.139,438.094,171.324,25.984,154.874
C08084=1061.097,-101.389,438.104,171.322,25.984,154.874
C08085=1061.091,-101.639,438.114,171.320,25.983,154.874
C08086=1061.084,-101.888,438.124,171.318,25.981,154.874
C08087=1061.079,-102.139,438.134,171.317,25.980,154.874
C08088=1061.073,-102.388,438.144,171.315,25.979,154.874
C08089=1061.066,-102.638,438.154,171.313,25.978,154.874
C08090=1061.060,-102.888,438.165,171.311,25.977,154.874
C08091=1061.054,-103.138,438.175,171.309,25.976,154.874
C08092=1061.048,-103.387,438.184,171.308,25.975,154.874
C08093=1061.042,-103.637,438.195,171.305,25.974,154.874
C08094=1061.036,-103.887,438.205,171.303,25.972,154.874
C08095=1061.029,-104.136,438.215,171.302,25.971,154.874
C08096=1061.023,-104.386,438.225,171.300,25.971,154.874
C08097=1061.018,-104.636,438.235,171.298,25.969,154.874
C08098=1061.011,-104.885,438.245,171.296,25.968,154.874
C08099=1061.005,-105.135,438.255,171.294,25.967,154.874
C08100=1061.000,-105.385,438.265,171.293,25.966,154.874
C08101=1060.993,-105.634,438.275,171.291,25.965,154.874
C08102=1060.986,-105.884,438.285,171.289,25.964,154.874
C08103=1060.980,-106.134,438.295,171.287,25.963,154.874
C08104=1060.974,-106.384,438.305,171.285,25.962,154.874
C08105=1060.968,-106.634,438.315,171.284,25.961,154.874
C08106=1060.962,-106.883,438.325,171.282,25.960,154.874
C08107=1060.956,-107.133,438.334,171.280,25.959,154.874
C08108=1060.950,-107.383,438.345,171.278,25.958,154.874
C08109=1060.944,-107.632,438.355,171.277,25.957,154.874
C08110=1060.938,-107.882,438.364,171.274,25.956,154.874
C08111=1060.932,-108.132,438.374,171.272,25.955,154.874
C08112=1060.925,-108.381,438.384,171.270,25.954,154.874
C08113=1060.919,-108.631,438.394,171.269,25.953,154.874
C08114=1060.913,-108.881,438.403,171.267,25.952,154.874
C08115=1060.907,-109.131,438.413,171.265,25.951,154.874
C08116=1060.901,-109.380,438.424,171.263,25.950,154.874
C08117=1060.895,-109.630,438.433,171.261,25.949,154.874
C08118=1060.889,-109.880,438.443,171.260,25.949,154.874
C08119=1060.882,-110.129,438.452,171.258,25.947,154.874
C08120=1060.876,-110.379,438.462,171.256,25.947,154.874
C08121=1060.870,-110.628,438.472,171.254,25.946,154.874
C08122=1060.864,-110.878,438.482,171.252,25.944,154.874
C08123=1060.857,-111.128,438.491,171.251,25.944,154.875
C08124=1060.851,-111.378,438.501,171.249,25.943,154.875
C08125=1060.846,-111.628,438.511,171.247,25.942,154.875
C08126=1060.840,-111.878,438.521,171.245,25.941,154.875
C08127=1060.834,-112.128,438.530,171.242,25.940,154.875
C08128=1060.827,-112.377,438.540,171.241,25.939,154.875
C08129=1060.821,-112.627,438.550,171.239,25.938,154.875
C08130=1060.815,-112.876,438.560,171.237,25.937,154.875
C08131=1060.809,-113.126,438.569,171.235,25.936,154.875
C08132=1060.802,-113.376,438.579,171.234,25.935,154.875
C08133=1060.796,-113.626,438.588,171.232,25.935,154.875
C08134=1060.790,-113.876,438.598,171.230,25.933,154.875
C08135=1060.784,-114.125,438.607,171.228,25.933,154.875
C08136=1060.777,-114.408,438.619,171.226,25.932,154.875
C08137=1060.770,-114.691,438.630,171.224,25.931,154.875
C08138=1060.763,-114.973,438.640,171.222,25.930,154.875
C08139=1060.756,-115.257,438.651,171.220,25.929,154.875
C08140=1060.750,-115.507,438.661,171.218,25.928,154.875
C08141=1060.744,-115.756,438.670,171.216,25.927,154.875
C08142=1060.738,-116.006,438.680,171.214,25.927,154.876
C08143=1060.732,-116.255,438.689,171.213,25.925,154.875
C08144=1060.726,-116.505,438.699,171.210,25.925,154.876
C08145=1060.720,-116.755,438.708,171.208,25.923,154.876
C08146=1060.714,-117.005,438.718,171.206,25.923,154.876
C08147=1060.707,-117.254,438.728,171.204,25.922,154.876
C08148=1060.701,-117.504,438.737,171.203,25.921,154.876
C08149=1060.694,-117.754,438.746,171.201,25.920,154.876
C08150=1060.688,-118.004,438.756,171.199,25.920,154.876
C08151=1060.682,-118.253,438.765,171.197,25.919,154.876
C08152=1060.676,-118.503,438.775,171.195,25.918,154.876
C08153=1060.670,-118.753,438.784,171.194,25.918,154.876
C08154=1060.664,-119.002,438.794,171.192,25.917,154.876
C08155=1060.658,-119.252,438.803,171.190,25.916,154.876
C08156=1060.652,-119.502,438.812,171.188,25.915,154.876
C08157=1060.646,-119.752,438.822,171.186,25.915,154.876
C08158=1060.640,-120.002,438.831,171.184,25.913,154.876
C08159=1060.634,-120.252,438.841,171.183,25.913,154.877
C08160=1060.627,-120.501,438.850,171.181,25.912,154.877
C08161=1060.620,-120.751,438.859,171.179,25.912,154.877
C08162=1060.615,-121.000,438.868,171.177,25.910,154.877
C08163=1060.609,-121.250,438.878,171.174,25.910,154.877
C08164=1060.603,-121.500,438.887,171.172,25.909,154.877
C08165=1060.597,-121.750,438.896,171.171,25.908,154.877
C08166=1060.591,-122.000,438.906,171.169,25.908,154.877
C08167=1060.584,-122.249,438.915,171.167,25.907,154.877
C08168=1060.577,-122.499,438.924,171.165,25.906,154.877
C08169=1060.572,-122.748,438.934,171.163,25.905,154.877
C08170=1060.566,-122.999,438.943,171.161,25.905,154.878
C08171=1060.560,-123.248,438.952,171.160,25.904,154.878
C08172=1060.554,-123.498,438.962,171.158,25.904,154.878
C08173=1060.547,-123.748,438.971,171.156,25.902,154.878
C08174=1060.541,-123.998,438.980,171.154,25.902,154.878
C08175=1060.535,-124.247,438.989,171.152,25.901,154.878
C08176=1060.529,-124.497,438.998,171.150,25.901,154.878
C08177=1060.523,-124.747,439.008,171.148,25.900,154.878
C08178=1060.516,-124.996,439.017,171.147,25.900,154.878
C08179=1060.510,-125.247,439.026,171.145,25.899,154.878
C08180=1060.505,-125.496,439.035,171.143,25.898,154.878
C08181=1060.498,-125.746,439.044,171.141,25.898,154.879
C08182=1060.492,-125.996,439.053,171.139,25.897,154.879
C08183=1060.486,-126.246,439.062,171.137,25.897,154.879
C08184=1060.480,-126.495,439.072,171.134,25.896,154.879
C08185=1060.474,-126.744,439.081,171.133,25.895,154.879
C08186=1060.467,-126.995,439.089,171.131,25.895,154.879
C08187=1060.461,-127.244,439.099,171.129,25.894,154.879
C08188=1060.455,-127.494,439.108,171.127,25.893,154.879
C08189=1060.448,-127.744,439.117,171.125,25.893,154.879
C08190=1060.444,-127.994,439.126,171.123,25.892,154.879
C08191=1060.439,-128.243,439.137,171.122,25.890,154.879
C08192=1060.436,-128.494,439.147,171.120,25.888,154.879
C08193=1060.435,-128.745,439.159,171.119,25.886,154.879
C08194=1060.435,-128.996,439.172,171.118,25.882,154.878
C08195=1060.436,-129.245,439.184,171.117,25.879,154.878
C08196=1060.439,-129.498,439.197,171.116,25.874,154.877
C08197=1060.443,-129.749,439.212,171.115,25.869,154.876
C08198=1060.450,-130.000,439.227,171.115,25.864,154.875
C08199=1060.456,-130.250,439.243,171.115,25.858,154.874
C08200=1060.078,-130.273,439.049,171.067,26.016,154.908
C08201=1060.071,-130.023,439.034,171.067,26.022,154.909
C08202=1060.065,-129.772,439.018,171.068,26.028,154.909
C08203=1060.061,-129.520,439.004,171.069,26.032,154.910
C08204=1060.057,-129.269,438.990,171.069,26.037,154.911
C08205=1060.056,-129.019,438.977,171.070,26.040,154.911
C08206=1060.056,-128.768,438.965,171.071,26.044,154.912
C08207=1060.057,-128.518,438.953,171.073,26.046,154.912
C08208=1060.060,-128.267,438.942,171.074,26.049,154.912
C08209=1060.064,-128.017,438.932,171.076,26.050,154.912
C08210=1060.069,-127.766,438.923,171.078,26.051,154.913
C08211=1060.076,-127.517,438.914,171.080,26.052,154.912
C08212=1060.082,-127.267,438.904,171.082,26.052,154.912
C08213=1060.087,-127.017,438.896,171.084,26.053,154.912
C08214=1060.094,-126.768,438.887,171.085,26.053,154.912
C08215=1060.100,-126.518,438.877,171.087,26.054,154.912
C08216=1060.106,-126.268,438.868,171.089,26.054,154.912
C08217=1060.112,-126.018,438.859,171.091,26.055,154.912
C08218=1060.119,-125.769,438.850,171.093,26.056,154.912
C08219=1060.125,-125.519,438.840,171.095,26.056,154.912
C08220=1060.131,-125.269,438.832,171.097,26.057,154.911
C08221=1060.137,-125.019,438.822,171.098,26.057,154.911
C08222=1060.144,-124.770,438.813,171.100,26.058,154.911
C08223=1060.149,-124.520,438.805,171.102,26.058,154.911
C08224=1060.155,-124.270,438.795,171.104,26.059,154.911
C08225=1060.161,-124.020,438.785,171.107,26.060,154.911
C08226=1060.168,-123.771,438.776,171.109,26.061,154.911
C08227=1060.174,-123.521,438.767,171.110,26.062,154.911
C08228=1060.180,-123.271,438.758,171.112,26.062,154.911
C08229=1060.186,-123.022,438.749,171.114,26.063,154.911
C08230=1060.192,-122.772,438.739,171.116,26.063,154.911
C08231=1060.198,-122.522,438.730,171.118,26.064,154.910
C08232=1060.205,-122.272,438.721,171.120,26.065,154.910
C08233=1060.211,-122.022,438.712,171.122,26.066,154.910
C08234=1060.217,-121.772,438.702,171.123,26.066,154.910
C08235=1060.223,-121.523,438.693,171.125,26.067,154.910
C08236=1060.229,-121.273,438.684,171.127,26.068,154.910
C08237=1060.235,-121.024,438.674,171.129,26.069,154.910
C08238=1060.241,-120.774,438.664,171.131,26.069,154.910
C08239=1060.247,-120.523,438.656,171.133,26.070,154.910
C08240=1060.254,-120.274,438.647,171.135,26.070,154.910
C08241=1060.260,-120.024,438.637,171.136,26.071,154.910
C08242=1060.266,-119.775,438.628,171.138,26.072,154.910
C08243=1060.272,-119.525,438.618,171.141,26.073,154.910
C08244=1060.278,-119.275,438.609,171.143,26.074,154.909
C08245=1060.284,-119.026,438.599,171.145,26.075,154.909
C08246=1060.290,-118.776,438.590,171.146,26.075,154.909
C08247=1060.297,-118.526,438.580,171.148,26.076,154.909
C08248=1060.303,-118.276,438.570,171.150,26.077,154.909
C08249=1060.309,-118.026,438.561,171.152,26.078,154.909
C08250=1060.316,-117.777,438.552,171.154,26.078,154.909
C08251=1060.322,-117.527,438.542,171.156,26.079,154.909
C08252=1060.327,-117.277,438.534,171.157,26.080,154.909
C08253=1060.333,-117.028,438.524,171.159,26.081,154.909
C08254=1060.340,-116.778,438.515,171.161,26.081,154.909
C08255=1060.346,-116.528,438.505,171.163,26.082,154.909
C08256=1060.352,-116.278,438.496,171.165,26.083,154.909
C08257=1060.358,-116.028,438.486,171.167,26.084,154.909
C08258=1060.364,-115.779,438.476,171.168,26.085,154.909
C08259=1060.371,-115.529,438.467,171.170,26.085,154.909
C08260=1060.377,-115.279,438.457,171.173,26.087,154.908
C08261=1060.383,-114.997,438.446,171.175,26.087,154.908
C08262=1060.391,-114.713,438.436,171.177,26.088,154.908
C08263=1060.397,-114.431,438.424,171.179,26.089,154.908
C08264=1060.404,-114.148,438.413,171.181,26.090,154.908
C08265=1060.410,-113.898,438.404,171.183,26.091,154.908
C08266=1060.417,-113.648,438.394,171.185,26.092,154.908
C08267=1060.423,-113.398,438.385,171.187,26.093,154.908
C08268=1060.429,-113.148,438.375,171.188,26.093,154.908
C08269=1060.435,-112.899,438.365,171.190,26.095,154.908
C08270=1060.442,-112.649,438.355,171.192,26.095,154.908
C08271=1060.448,-112.400,438.346,171.194,26.096,154.908
C08272=1060.454,-112.150,438.336,171.196,26.097,154.908
C08273=1060.460,-111.900,438.326,171.197,26.098,154.908
C08274=1060.466,-111.650,438.317,171.199,26.099,154.908
C08275=1060.472,-111.400,438.307,171.202,26.100,154.908
C08276=1060.478,-111.150,438.297,171.204,26.101,154.908
C08277=1060.484,-110.901,438.287,171.206,26.102,154.908
C08278=1060.491,-110.651,438.277,171.207,26.103,154.908
C08279=1060.497,-110.401,438.268,171.209,26.104,154.908
C08280=1060.503,-110.152,438.258,171.211,26.105,154.908
C08281=1060.509,-109.902,438.249,171.213,26.105,154.907
C08282=1060.516,-109.653,438.238,171.214,26.107,154.907
C08283=1060.522,-109.403,438.229,171.216,26.107,154.907
C08284=1060.527,-109.153,438.219,171.218,26.108,154.907
C08285=1060.533,-108.903,438.209,171.220,26.110,154.907
C08286=1060.540,-108.653,438.199,171.222,26.110,154.907
C08287=1060.546,-108.404,438.189,171.223,26.111,154.907
C08288=1060.552,-108.154,438.180,171.225,26.112,154.907
C08289=1060.558,-107.904,438.170,171.227,26.113,154.907
C08290=1060.565,-107.655,438.160,171.229,26.114,154.907
C08291=1060.571,-107.405,438.150,171.232,26.115,154.907
C08292=1060.576,-107.155,438.140,171.233,26.116,154.907
C08293=1060.583,-106.906,438.130,171.235,26.117,154.907
C08294=1060.589,-106.656,438.121,171.237,26.118,154.907
C08295=1060.595,-106.407,438.111,171.239,26.119,154.907
C08296=1060.601,-106.156,438.100,171.240,26.120,154.907
C08297=1060.607,-105.907,438.091,171.242,26.122,154.907
C08298=1060.613,-105.657,438.081,171.244,26.122,154.907
C08299=1060.620,-105.408,438.071,171.246,26.123,154.907
C08300=1060.626,-105.157,438.061,171.248,26.124,154.907
C08301=1060.632,-104.908,438.050,171.249,26.126,154.907
C08302=1060.638,-104.658,438.041,171.251,26.126,154.907
C08303=1060.644,-104.408,438.031,171.253,26.127,154.907
C08304=1060.650,-104.159,438.020,171.255,26.129,154.907
C08305=1060.656,-103.909,438.011,171.256,26.130,154.907
C08306=1060.663,-103.660,438.000,171.258,26.130,154.907
C08307=1060.668,-103.410,437.990,171.261,26.132,154.907
C08308=1060.674,-103.160,437.981,171.263,26.133,154.907
C08309=1060.681,-102.911,437.970,171.264,26.134,154.907
C08310=1060.686,-102.660,437.960,171.266,26.135,154.907
C08311=1060.693,-102.411,437.950,171.268,26.136,154.907
C08312=1060.700,-102.161,437.940,171.270,26.137,154.907
C08313=1060.705,-101.911,437.930,171.272,26.138,154.907
C08314=1060.711,-101.661,437.920,171.273,26.139,154.907
C08315=1060.718,-101.412,437.910,171.275,26.141,154.907
C08316=1060.723,-101.162,437.899,171.277,26.142,154.907
C08317=1060.730,-100.912,437.890,171.279,26.143,154.907
C08318=1060.736,-100.663,437.879,171.280,26.143,154.907
C08319=1060.742,-100.412,437.869,171.282,26.145,154.907
C08320=1060.749,-100.163,437.858,171.284,26.146,154.907
C08321=1060.755,-99.913,437.849,171.286,26.147,154.907
C08322=1060.760,-99.664,437.838,171.288,26.148,154.907
C08323=1060.767,-99.414,437.828,171.290,26.150,154.907
C08324=1060.773,-99.165,437.818,171.292,26.151,154.907
C08325=1060.780,-98.880,437.806,171.294,26.152,154.907
C08326=1060.787,-98.596,437.794,171.295,26.153,154.907
C08327=1060.794,-98.311,437.783,171.298,26.155,154.907
C08328=1060.801,-98.027,437.771,171.300,26.156,154.907
C08329=1060.807,-97.776,437.761,171.302,26.157,154.907
C08330=1060.814,-97.527,437.751,171.303,26.158,154.907
C08331=1060.819,-97.277,437.741,171.305,26.159,154.907
C08332=1060.825,-97.027,437.730,171.307,26.160,154.907
C08333=1060.831,-96.778,437.720,171.309,26.162,154.907
C08334=1060.837,-96.528,437.709,171.310,26.163,154.907
C08335=1060.844,-96.278,437.699,171.312,26.164,154.907
C08336=1060.850,-96.028,437.688,171.315,26.165,154.907
C08337=1060.856,-95.779,437.678,171.316,26.167,154.907
C08338=1060.862,-95.529,437.667,171.318,26.168,154.907
C08339=1060.867,-95.279,437.657,171.320,26.169,154.907
C08340=1060.874,-95.030,437.647,171.322,26.171,154.907
C08341=1060.880,-94.779,437.636,171.323,26.172,154.907
C08342=1060.886,-94.530,437.626,171.325,26.173,154.907
C08343=1060.892,-94.281,437.615,171.327,26.174,154.907
C08344=1060.898,-94.031,437.606,171.329,26.175,154.907
C08345=1060.904,-93.781,437.595,171.330,26.176,154.907
C08346=1060.910,-93.531,437.584,171.332,26.178,154.907
C08347=1060.917,-93.282,437.573,171.334,26.179,154.908
C08348=1060.922,-93.032,437.563,171.335,26.181,154.908
C08349=1060.929,-92.783,437.553,171.337,26.182,154.908
C08350=1060.935,-92.533,437.542,171.339,26.183,154.908
C08351=1060.940,-92.282,437.531,171.341,26.184,154.908
C08352=1060.947,-92.033,437.521,171.343,26.186,154.908
C08353=1060.953,-91.784,437.510,171.345,26.187,154.908
C08354=1060.959,-91.534,437.499,171.347,26.188,154.908
C08355=1060.965,-91.284,437.489,171.348,26.190,154.908
C08356=1060.971,-91.034,437.479,171.350,26.191,154.908
C08357=1060.977,-90.785,437.468,171.352,26.192,154.908
C08358=1060.984,-90.535,437.457,171.354,26.194,154.908
C08359=1060.989,-90.285,437.446,171.355,26.195,154.908
C08360=1060.996,-90.036,437.437,171.357,26.196,154.908
C08361=1061.001,-89.786,437.426,171.359,26.197,154.908
C08362=1061.008,-89.536,437.414,171.360,26.199,154.908
C08363=1061.014,-89.287,437.404,171.362,26.200,154.908
C08364=1061.020,-89.037,437.393,171.364,26.201,154.908
C08365=1061.027,-88.787,437.383,171.366,26.202,154.908
C08366=1061.032,-88.537,437.372,171.367,26.204,154.908
C08367=1061.038,-88.288,437.362,171.369,26.205,154.908
C08368=1061.045,-88.038,437.351,171.372,26.207,154.908
C08369=1061.051,-87.788,437.340,171.374,26.208,154.908
C08370=1061.057,-87.539,437.329,171.375,26.210,154.909
C08371=1061.063,-87.290,437.319,171.377,26.211,154.909
C08372=1061.069,-87.040,437.308,171.379,26.212,154.909
C08373=1061.075,-86.790,437.297,171.380,26.214,154.909
C08374=1061.082,-86.540,437.287,171.382,26.215,154.909
C08375=1061.088,-86.290,437.276,171.384,26.216,154.909
C08376=1061.093,-86.041,437.265,171.386,26.217,154.909
C08377=1061.101,-85.791,437.254,171.387,26.219,154.909
C08378=1061.106,-85.541,437.244,171.389,26.220,154.909
C08379=1061.112,-85.292,437.233,171.391,26.221,154.909
C08380=1061.118,-85.042,437.221,171.392,26.223,154.909
C08381=1061.125,-84.792,437.211,171.394,26.224,154.909
C08382=1061.131,-84.543,437.200,171.396,26.225,154.909
C08383=1061.137,-84.293,437.189,171.397,26.227,154.909
C08384=1061.143,-84.044,437.179,171.400,26.229,154.909
C08385=1061.150,-83.793,437.168,171.402,26.230,154.909
C08386=1061.155,-83.544,437.157,171.403,26.232,154.909
C08387=1061.162,-83.295,437.146,171.405,26.233,154.909
C08388=1061.168,-83.045,437.135,171.407,26.235,154.910
C08389=1061.175,-82.763,437.123,171.409,26.236,154.910
C08390=1061.182,-82.480,437.110,171.410,26.237,154.910
C08391=1061.189,-82.197,437.098,171.413,26.239,154.910
C08392=1061.196,-81.916,437.086,171.415,26.241,154.910
C08393=1061.202,-81.665,437.075,171.416,26.242,154.910
C08394=1061.208,-81.416,437.064,171.418,26.244,154.910
C08395=1061.215,-81.166,437.054,171.420,26.245,154.910
C08396=1061.221,-80.917,437.042,171.421,26.246,154.910
C08397=1061.228,-80.667,437.031,171.423,26.248,154.910
C08398=1061.234,-80.418,437.020,171.426,26.249,154.910
C08399=1061.240,-80.168,437.010,171.427,26.251,154.910
C08400=1061.246,-79.918,436.998,171.429,26.252,154.910
C08401=1061.252,-79.669,436.987,171.431,26.254,154.910
C08402=1061.258,-79.418,436.976,171.433,26.255,154.910
C08403=1061.264,-79.169,436.965,171.434,26.257,154.911
C08404=1061.270,-78.919,436.954,171.436,26.258,154.911
C08405=1061.276,-78.670,436.943,171.438,26.260,154.911
C08406=1061.283,-78.420,436.932,171.439,26.261,154.911
C08407=1061.289,-78.170,436.921,171.441,26.262,154.911
C08408=1061.295,-77.921,436.910,171.443,26.264,154.911
C08409=1061.301,-77.671,436.899,171.444,26.265,154.911
C08410=1061.307,-77.421,436.888,171.446,26.267,154.911
C08411=1061.314,-77.172,436.876,171.448,26.268,154.911
C08412=1061.319,-76.922,436.865,171.449,26.270,154.911
C08413=1061.326,-76.672,436.854,171.451,26.272,154.912
C08414=1061.331,-76.423,436.843,171.453,26.273,154.912
C08415=1061.338,-76.173,436.831,171.454,26.275,154.912
C08416=1061.344,-75.923,436.820,171.457,26.276,154.912
C08417=1061.350,-75.673,436.809,171.459,26.278,154.912
C08418=1061.356,-75.424,436.798,171.460,26.280,154.912
C08419=1061.362,-75.174,436.786,171.462,26.281,154.912
C08420=1061.368,-74.925,436.775,171.464,26.283,154.912
C08421=1061.375,-74.675,436.764,171.465,26.284,154.912
C08422=1061.380,-74.425,436.753,171.467,26.286,154.912
C08423=1061.387,-74.175,436.741,171.469,26.287,154.912
C08424=1061.393,-73.926,436.730,171.470,26.289,154.913
C08425=1061.399,-73.676,436.719,171.472,26.290,154.913
C08426=1061.405,-73.427,436.707,171.474,26.292,154.913
C08427=1061.411,-73.177,436.696,171.475,26.294,154.913
C08428=1061.417,-72.927,436.685,171.477,26.295,154.913
C08429=1061.423,-72.677,436.673,171.479,26.297,154.913
C08430=1061.429,-72.428,436.662,171.480,26.299,154.913
C08431=1061.435,-72.178,436.651,171.482,26.300,154.913
C08432=1061.441,-71.929,436.639,171.484,26.302,154.913
C08433=1061.447,-71.679,436.628,171.485,26.304,154.914
C08434=1061.453,-71.429,436.616,171.487,26.305,154.914
C08435=1061.459,-71.180,436.605,171.489,26.307,154.914
C08436=1061.465,-70.930,436.594,171.491,26.309,154.914
C08437=1061.471,-70.681,436.582,171.493,26.311,154.914
C08438=1061.477,-70.430,436.570,171.494,26.312,154.914
C08439=1061.483,-70.182,436.558,171.496,26.314,154.914
C08440=1061.489,-69.931,436.547,171.498,26.315,154.914
C08441=1061.495,-69.681,436.536,171.499,26.317,154.915
C08442=1061.501,-69.432,436.524,171.501,26.319,154.915
C08443=1061.507,-69.182,436.513,171.503,26.321,154.915
C08444=1061.513,-68.933,436.501,171.504,26.322,154.915
C08445=1061.519,-68.683,436.490,171.506,26.324,154.915
C08446=1061.525,-68.434,436.478,171.508,26.325,154.915
C08447=1061.531,-68.183,436.466,171.509,26.327,154.915
C08448=1061.537,-67.934,436.455,171.511,26.329,154.915
C08449=1061.543,-67.684,436.443,171.513,26.331,154.916
C08450=1061.550,-67.435,436.431,171.514,26.332,154.916
C08451=1061.555,-67.185,436.420,171.516,26.334,154.916
C08452=1061.562,-66.935,436.408,171.517,26.336,154.916
C08453=1061.568,-66.655,436.396,171.520,26.338,154.916
C08454=1061.575,-66.375,436.383,171.522,26.340,154.916
C08455=1061.582,-66.096,436.369,171.523,26.341,154.916
C08456=1061.589,-65.816,436.356,171.526,26.344,154.917
C08457=1061.595,-65.565,436.345,171.527,26.346,154.917
C08458=1061.601,-65.316,436.333,171.529,26.347,154.917
C08459=1061.607,-65.066,436.322,171.531,26.349,154.917
C08460=1061.613,-64.817,436.309,171.532,26.350,154.917
C08461=1061.619,-64.566,436.298,171.534,26.352,154.917
C08462=1061.625,-64.317,436.286,171.536,26.354,154.917
C08463=1061.632,-64.068,436.274,171.537,26.356,154.917
C08464=1061.637,-63.818,436.263,171.539,26.357,154.918
C08465=1061.644,-63.569,436.251,171.541,26.359,154.918
C08466=1061.650,-63.319,436.239,171.542,26.361,154.918
C08467=1061.655,-63.069,436.227,171.544,26.363,154.918
C08468=1061.662,-62.820,436.216,171.546,26.364,154.918
C08469=1061.668,-62.570,436.204,171.547,26.366,154.918
C08470=1061.674,-62.321,436.193,171.549,26.368,154.918
C08471=1061.680,-62.071,436.180,171.550,26.370,154.919
C08472=1061.687,-61.821,436.168,171.552,26.371,154.919
C08473=1061.692,-61.572,436.157,171.554,26.373,154.919
C08474=1061.698,-61.322,436.145,171.555,26.375,154.919
C08475=1061.705,-61.072,436.133,171.557,26.377,154.919
C08476=1061.711,-60.822,436.122,171.559,26.378,154.919
C08477=1061.717,-60.573,436.109,171.560,26.380,154.919
C08478=1061.723,-60.323,436.097,171.562,26.382,154.920
C08479=1061.730,-60.073,436.086,171.563,26.384,154.920
C08480=1061.735,-59.824,436.074,171.566,26.386,154.920
C08481=1061.742,-59.574,436.062,171.568,26.388,154.920
C08482=1061.748,-59.325,436.050,171.569,26.390,154.920
C08483=1061.754,-59.074,436.038,171.571,26.391,154.920
C08484=1061.760,-58.825,436.027,171.573,26.393,154.921
C08485=1061.767,-58.576,436.015,171.574,26.395,154.921
C08486=1061.772,-58.326,436.002,171.576,26.397,154.921
C08487=1061.779,-58.076,435.990,171.577,26.398,154.921
C08488=1061.785,-57.827,435.979,171.579,26.400,154.921
C08489=1061.791,-57.577,435.967,171.581,26.402,154.921
C08490=1061.797,-57.327,435.955,171.582,26.403,154.921
C08491=1061.804,-57.078,435.943,171.584,26.405,154.922
C08492=1061.809,-56.829,435.931,171.586,26.407,154.922
C08493=1061.816,-56.579,435.919,171.587,26.409,154.922
C08494=1061.822,-56.328,435.907,171.589,26.411,154.922
C08495=1061.828,-56.079,435.895,171.590,26.413,154.922
C08496=1061.835,-55.829,435.883,171.592,26.415,154.922
C08497=1061.840,-55.580,435.871,171.594,26.416,154.923
C08498=1061.847,-55.331,435.859,171.595,26.418,154.923
C08499=1061.854,-55.081,435.847,171.597,26.420,154.923
C08500=1061.859,-54.831,435.834,171.599,26.421,154.923
C08501=1061.866,-54.582,435.822,171.600,26.423,154.923
C08502=1061.872,-54.331,435.810,171.602,26.426,154.923
C08503=1061.878,-54.082,435.799,171.603,26.427,154.923
C08504=1061.884,-53.833,435.787,171.605,26.429,154.924
C08505=1061.894,-53.450,435.768,171.608,26.432,154.924
C08506=1061.903,-53.067,435.750,171.611,26.435,154.924
C08507=1061.913,-52.684,435.731,171.613,26.438,154.924
C08508=1061.922,-52.301,435.712,171.616,26.440,154.925
C08509=1061.929,-52.052,435.700,171.617,26.442,154.925
C08510=1061.935,-51.802,435.688,171.619,26.444,154.925
C08511=1061.941,-51.552,435.676,171.621,26.446,154.925
C08512=1061.948,-51.303,435.664,171.622,26.448,154.925
C08513=1061.958,-50.908,435.645,171.625,26.450,154.925
C08514=1061.967,-50.513,435.625,171.628,26.454,154.926
C08515=1061.978,-50.117,435.606,171.630,26.457,154.926
C08516=1061.987,-49.722,435.586,171.633,26.460,154.926
C08517=1061.993,-49.472,435.574,171.634,26.461,154.926
C08518=1061.999,-49.223,435.561,171.636,26.464,154.927
C08519=1062.005,-48.973,435.549,171.638,26.466,154.927
C08520=1062.010,-48.723,435.536,171.639,26.468,154.927
C08521=1062.017,-48.474,435.524,171.641,26.470,154.927
C08522=1062.023,-48.224,435.511,171.642,26.471,154.927
C08523=1062.029,-47.975,435.499,171.644,26.474,154.928
C08524=1062.035,-47.726,435.487,171.646,26.475,154.928
C08525=1062.041,-47.476,435.474,171.647,26.478,154.928
C08526=1062.047,-47.226,435.462,171.649,26.479,154.928
C08527=1062.053,-46.976,435.449,171.650,26.482,154.928
C08528=1062.060,-46.726,435.437,171.652,26.483,154.929
C08529=1062.066,-46.477,435.424,171.654,26.485,154.929
C08530=1062.072,-46.227,435.412,171.655,26.488,154.929
C08531=1062.078,-45.977,435.399,171.657,26.489,154.929
C08532=1062.084,-45.728,435.387,171.658,26.492,154.929
C08533=1062.090,-45.479,435.375,171.660,26.493,154.930
C08534=1062.096,-45.229,435.362,171.661,26.496,154.930
C08535=1062.102,-44.980,435.349,171.663,26.497,154.930
C08536=1062.108,-44.730,435.337,171.665,26.499,154.930
C08537=1062.114,-44.480,435.325,171.666,26.501,154.930
C08538=1062.120,-44.230,435.312,171.668,26.503,154.931
C08539=1062.126,-43.981,435.299,171.669,26.505,154.931
C08540=1062.133,-43.731,435.287,171.671,26.507,154.931
C08541=1062.139,-43.481,435.274,171.673,26.509,154.931
C08542=1062.145,-43.232,435.262,171.674,26.511,154.931
C08543=1062.151,-42.982,435.248,171.676,26.514,154.932
C08544=1062.158,-42.733,435.236,171.677,26.515,154.932
C08545=1062.164,-42.483,435.224,171.679,26.518,154.932
C08546=1062.170,-42.234,435.211,171.681,26.519,154.932
C08547=1062.176,-41.984,435.198,171.682,26.522,154.932
C08548=1062.182,-41.735,435.186,171.685,26.524,154.933
C08549=1062.188,-41.485,435.174,171.686,26.526,154.933
C08550=1062.194,-41.236,435.161,171.688,26.528,154.933
C08551=1062.200,-40.986,435.148,171.689,26.530,154.933
C08552=1062.206,-40.736,435.136,171.691,26.532,154.933
C08553=1062.213,-40.487,435.123,171.693,26.534,154.934
C08554=1062.219,-40.237,435.110,171.694,26.536,154.934
C08555=1062.225,-39.988,435.097,171.696,26.538,154.934
C08556=1062.231,-39.738,435.084,171.697,26.540,154.934
C08557=1062.237,-39.488,435.072,171.699,26.542,154.934
C08558=1062.244,-39.239,435.059,171.701,26.544,154.935
C08559=1062.250,-38.989,435.047,171.702,26.546,154.935
C08560=1062.256,-38.739,435.034,171.704,26.548,154.935
C08561=1062.262,-38.489,435.020,171.705,26.550,154.935
C08562=1062.268,-38.239,435.008,171.707,26.552,154.935
C08563=1062.274,-37.990,434.995,171.708,26.554,154.936
C08564=1062.280,-37.740,434.982,171.710,26.557,154.936
C08565=1062.287,-37.491,434.969,171.712,26.558,154.936
C08566=1062.292,-37.242,434.957,171.713,26.561,154.936
C08567=1062.298,-36.993,434.943,171.715,26.563,154.937
C08568=1062.304,-36.743,434.931,171.716,26.565,154.937
C08569=1062.310,-36.493,434.918,171.718,26.567,154.937
C08570=1062.317,-36.243,434.905,171.719,26.569,154.937
C08571=1062.323,-35.993,434.892,171.721,26.571,154.937
C08572=1062.329,-35.744,434.879,171.723,26.573,154.938
C08573=1062.335,-35.494,434.866,171.724,26.576,154.938
C08574=1062.341,-35.245,434.853,171.726,26.577,154.938
C08575=1062.347,-34.995,434.840,171.727,26.580,154.938
C08576=1062.353,-34.745,434.827,171.729,26.582,154.939
C08577=1062.359,-34.467,434.812,171.730,26.584,154.939
C08578=1062.367,-34.189,434.798,171.732,26.587,154.939
C08579=1062.373,-33.910,434.784,171.733,26.589,154.939
C08580=1062.380,-33.632,434.769,171.736,26.592,154.940
C08581=1062.386,-33.383,434.756,171.738,26.593,154.940
C08582=1062.392,-33.133,434.743,171.739,26.596,154.940
C08583=1062.398,-32.883,434.730,171.741,26.598,154.940
C08584=1062.405,-32.634,434.717,171.742,26.600,154.941
C08585=1062.411,-32.384,434.704,171.744,26.602,154.941
C08586=1062.417,-32.135,434.691,171.745,26.604,154.941
C08587=1062.422,-31.885,434.678,171.747,26.607,154.941
C08588=1062.428,-31.636,434.665,171.749,26.608,154.941
C08589=1062.434,-31.386,434.651,171.750,26.611,154.942
C08590=1062.441,-31.136,434.639,171.752,26.613,154.942
C08591=1062.447,-30.887,434.625,171.753,26.615,154.942
C08592=1062.453,-30.637,434.612,171.755,26.617,154.942
C08593=1062.459,-30.387,434.599,171.756,26.619,154.943
C08594=1062.465,-30.138,434.586,171.758,26.622,154.943
C08595=1062.472,-29.889,434.573,171.759,26.624,154.943
C08596=1062.478,-29.639,434.560,171.761,26.626,154.943
C08597=1062.484,-29.390,434.547,171.763,26.628,154.944
C08598=1062.491,-29.140,434.533,171.764,26.630,154.944
C08599=1062.497,-28.890,434.520,171.765,26.632,154.944
C08600=1062.502,-28.640,434.507,171.766,26.634,154.944
C08601=1062.508,-28.391,434.494,171.768,26.636,154.945
C08602=1062.514,-28.142,434.480,171.769,26.639,154.945
C08603=1062.520,-27.892,434.468,171.771,26.641,154.945
C08604=1062.527,-27.642,434.454,171.773,26.643,154.945
C08605=1062.533,-27.393,434.441,171.774,26.645,154.946
C08606=1062.540,-27.143,434.428,171.776,26.647,154.946
C08607=1062.546,-26.894,434.414,171.777,26.649,154.946
C08608=1062.551,-26.644,434.401,171.779,26.651,154.946
C08609=1062.557,-26.395,434.388,171.780,26.654,154.946
C08610=1062.564,-26.145,434.374,171.782,26.656,154.947
C08611=1062.570,-25.895,434.361,171.784,26.658,154.947
C08612=1062.576,-25.646,434.347,171.785,26.660,154.947
C08613=1062.582,-25.396,434.335,171.787,26.663,154.948
C08614=1062.588,-25.147,434.321,171.788,26.665,154.948
C08615=1062.593,-24.897,434.308,171.790,26.667,154.948
C08616=1062.600,-24.647,434.294,171.791,26.670,154.948
C08617=1062.606,-24.398,434.281,171.793,26.672,154.949
C08618=1062.612,-24.148,434.267,171.794,26.674,154.949
C08619=1062.618,-23.899,434.254,171.796,26.676,154.949
C08620=1062.624,-23.649,434.241,171.798,26.678,154.949
C08621=1062.629,-23.400,434.227,171.799,26.681,154.950
C08622=1062.636,-23.150,434.213,171.801,26.683,154.950
C08623=1062.642,-22.900,434.200,171.802,26.685,154.950
C08624=1062.648,-22.651,434.186,171.804,26.687,154.950
C08625=1062.654,-22.402,434.173,171.805,26.690,154.951
C08626=1062.660,-22.152,434.160,171.807,26.692,154.951
C08627=1062.666,-21.902,434.146,171.808,26.694,154.951
C08628=1062.673,-21.653,434.132,171.810,26.697,154.951
C08629=1062.679,-21.403,434.119,171.811,26.699,154.952
C08630=1062.684,-21.154,434.105,171.813,26.701,154.952
C08631=1062.691,-20.904,434.092,171.815,26.704,154.952
C08632=1062.697,-20.655,434.078,171.816,26.706,154.952
C08633=1062.703,-20.405,434.064,171.818,26.708,154.953
C08634=1062.709,-20.156,434.051,171.819,26.710,154.953
C08635=1062.715,-19.906,434.037,171.821,26.712,154.953
C08636=1062.721,-19.656,434.024,171.822,26.715,154.953
C08637=1062.728,-19.407,434.010,171.824,26.717,154.954
C08638=1062.733,-19.157,433.997,171.825,26.719,154.954
C08639=1062.740,-18.907,433.983,171.827,26.721,154.954
C08640=1062.746,-18.658,433.970,171.829,26.724,154.954
C08641=1062.752,-18.379,433.954,171.830,26.726,154.955
C08642=1062.759,-18.100,433.938,171.832,26.729,154.955
C08643=1062.766,-17.820,433.924,171.833,26.731,154.955
C08644=1062.773,-17.541,433.908,171.835,26.733,154.956
C08645=1062.779,-17.292,433.895,171.836,26.736,154.956
C08646=1062.785,-17.043,433.881,171.838,26.738,154.956
C08647=1062.791,-16.793,433.867,171.839,26.740,154.956
C08648=1062.798,-16.543,433.853,171.841,26.743,154.957
C08649=1062.804,-16.294,433.840,171.842,26.745,154.957
C08650=1062.810,-16.045,433.827,171.844,26.747,154.957
C08651=1062.816,-15.794,433.812,171.845,26.750,154.958
C08652=1062.822,-15.545,433.799,171.847,26.752,154.958
C08653=1062.828,-15.295,433.785,171.849,26.754,154.958
C08654=1062.835,-15.046,433.771,171.850,26.756,154.958
C08655=1062.840,-14.797,433.757,171.852,26.759,154.959
C08656=1062.847,-14.547,433.744,171.853,26.761,154.959
C08657=1062.853,-14.297,433.730,171.855,26.764,154.959
C08658=1062.859,-14.048,433.716,171.856,26.766,154.960
C08659=1062.864,-13.798,433.702,171.858,26.769,154.960
C08660=1062.871,-13.549,433.687,171.859,26.771,154.960
C08661=1062.877,-13.299,433.674,171.861,26.773,154.960
C08662=1062.882,-13.050,433.660,171.862,26.775,154.961
C08663=1062.888,-12.799,433.646,171.864,26.778,154.961
C08664=1062.895,-12.551,433.632,171.865,26.780,154.961
C08665=1062.900,-12.301,433.618,171.867,26.783,154.962
C08666=1062.907,-12.051,433.605,171.868,26.785,154.962
C08667=1062.913,-11.802,433.591,171.870,26.787,154.962
C08668=1062.919,-11.553,433.576,171.872,26.790,154.962
C08669=1062.925,-11.303,433.563,171.872,26.792,154.963
C08670=1062.931,-11.053,433.549,171.874,26.794,154.963
C08671=1062.936,-10.804,433.535,171.875,26.796,154.963
C08672=1062.943,-10.554,433.520,171.877,26.799,154.963
C08673=1062.949,-10.305,433.507,171.878,26.802,154.964
C08674=1062.956,-10.055,433.493,171.880,26.804,154.964
C08675=1062.962,-9.806,433.478,171.881,26.806,154.964
C08676=1062.967,-9.556,433.464,171.883,26.808,154.965
C08677=1062.974,-9.306,433.451,171.884,26.811,154.965
C08678=1062.980,-9.057,433.436,171.886,26.813,154.965
C08679=1062.986,-8.807,433.422,171.888,26.815,154.965
C08680=1062.992,-8.558,433.409,171.889,26.818,154.966
C08681=1062.998,-8.309,433.394,171.891,26.820,154.966
C08682=1063.004,-8.058,433.380,171.892,26.823,154.966
C08683=1063.010,-7.810,433.366,171.894,26.825,154.967
C08684=1063.016,-7.560,433.352,171.895,26.827,154.967
C08685=1063.022,-7.310,433.338,171.897,26.830,154.967
C08686=1063.029,-7.061,433.324,171.898,26.832,154.967
C08687=1063.034,-6.811,433.310,171.900,26.835,154.968
C08688=1063.040,-6.562,433.295,171.901,26.837,154.968
C08689=1063.047,-6.312,433.281,171.903,26.839,154.968
C08690=1063.052,-6.063,433.268,171.903,26.841,154.969
C08691=1063.059,-5.813,433.253,171.905,26.844,154.969
C08692=1063.065,-5.564,433.239,171.907,26.846,154.969
C08693=1063.071,-5.314,433.224,171.908,26.849,154.970
C08694=1063.077,-5.064,433.211,171.910,26.851,154.970
C08695=1063.083,-4.815,433.196,171.911,26.853,154.970
C08696=1063.090,-4.565,433.182,171.913,26.856,154.970
C08697=1063.096,-4.316,433.167,171.914,26.858,154.971
C08698=1063.101,-4.066,433.154,171.916,26.860,154.971
C08699=1063.109,-3.817,433.139,171.917,26.863,154.971
C08700=1063.114,-3.567,433.125,171.919,26.865,154.972
C08701=1063.120,-3.318,433.110,171.920,26.868,154.972
C08702=1063.126,-3.068,433.097,171.922,26.870,154.972
C08703=1063.132,-2.818,433.082,171.923,26.873,154.973
C08704=1063.138,-2.569,433.068,171.925,26.875,154.973
C08705=1063.145,-2.288,433.051,171.926,26.878,154.973
C08706=1063.152,-2.007,433.036,171.928,26.880,154.973
C08707=1063.158,-1.727,433.019,171.929,26.883,154.974
C08708=1063.165,-1.447,433.002,171.931,26.886,154.974
C08709=1063.171,-1.196,432.988,171.932,26.888,154.974
C08710=1063.177,-0.947,432.974,171.934,26.891,154.975
C08711=1063.183,-0.697,432.959,171.935,26.894,154.975
C08712=1063.189,-0.448,432.945,171.937,26.896,154.975
C08713=1063.194,-0.199,432.930,171.938,26.899,154.976
C08714=1063.201,0.051,432.916,171.940,26.901,154.976
C08715=1063.206,0.300,432.901,171.941,26.903,154.976
C08716=1063.213,0.550,432.886,171.943,26.906,154.977
C08717=1063.218,0.799,432.873,171.944,26.908,154.977
C08718=1063.225,1.049,432.858,171.946,26.911,154.977
C08719=1063.230,1.298,432.843,171.947,26.914,154.978
C08720=1063.236,1.548,432.829,171.949,26.916,154.978
C08721=1063.242,1.797,432.814,171.950,26.918,154.978
C08722=1063.249,2.047,432.799,171.951,26.921,154.979
C08723=1063.255,2.297,432.785,171.953,26.923,154.979
C08724=1063.260,2.546,432.770,171.954,26.926,154.979
C08725=1063.267,2.796,432.756,171.956,26.928,154.980
C08726=1063.273,3.045,432.741,171.957,26.930,154.980
C08727=1063.279,3.295,432.727,171.959,26.933,154.980
C08728=1063.285,3.544,432.712,171.960,26.936,154.980
C08729=1063.291,3.793,432.697,171.962,26.938,154.981
C08730=1063.297,4.042,432.683,171.963,26.941,154.981
C08731=1063.303,4.293,432.668,171.965,26.943,154.981
C08732=1063.309,4.542,432.654,171.966,26.945,154.982
C08733=1063.315,4.791,432.639,171.968,26.948,154.982
C08734=1063.321,5.041,432.624,171.969,26.950,154.982
C08735=1063.327,5.290,432.609,171.970,26.952,154.983
C08736=1063.333,5.540,432.595,171.971,26.955,154.983
C08737=1063.339,5.789,432.581,171.973,26.958,154.983
C08738=1063.345,6.039,432.566,171.975,26.960,154.984
C08739=1063.352,6.288,432.551,171.976,26.963,154.984
C08740=1063.357,6.537,432.536,171.978,26.965,154.984
C08741=1063.364,6.787,432.521,171.979,26.968,154.985
C08742=1063.369,7.037,432.507,171.981,26.970,154.985
C08743=1063.376,7.286,432.492,171.982,26.972,154.985
C08744=1063.381,7.536,432.477,171.984,26.975,154.986
C08745=1063.387,7.785,432.462,171.985,26.978,154.986
C08746=1063.394,8.035,432.447,171.987,26.980,154.986
C08747=1063.400,8.285,432.432,171.988,26.983,154.986
C08748=1063.406,8.533,432.418,171.989,26.985,154.987
C08749=1063.412,8.783,432.403,171.990,26.988,154.987
C08750=1063.418,9.033,432.389,171.992,26.990,154.987
C08751=1063.424,9.282,432.374,171.993,26.992,154.988
C08752=1063.430,9.532,432.359,171.995,26.995,154.988
C08753=1063.437,9.782,432.344,171.996,26.997,154.988
C08754=1063.442,10.031,432.329,171.998,27.000,154.989
C08755=1063.449,10.280,432.315,172.000,27.002,154.989
C08756=1063.455,10.530,432.300,172.001,27.005,154.989
C08757=1063.460,10.779,432.284,172.003,27.008,154.990
C08758=1063.467,11.029,432.269,172.004,27.010,154.990
C08759=1063.473,11.279,432.254,172.006,27.012,154.990
C08760=1063.479,11.527,432.240,172.007,27.015,154.991
C08761=1063.485,11.777,432.225,172.008,27.017,154.991
C08762=1063.492,12.027,432.210,172.009,27.019,154.991
C08763=1063.498,12.276,432.195,172.011,27.022,154.992
C08764=1063.504,12.525,432.180,172.012,27.024,154.992
C08765=1063.510,12.775,432.166,172.014,27.027,154.992
C08766=1063.517,13.025,432.151,172.015,27.030,154.993
C08767=1063.522,13.274,432.135,172.017,27.032,154.993
C08768=1063.528,13.524,432.120,172.018,27.035,154.993
C08769=1063.535,13.806,432.103,172.020,27.038,154.994
C08770=1063.542,14.089,432.087,172.021,27.040,154.994
C08771=1063.550,14.371,432.070,172.023,27.043,154.994
C08772=1063.556,14.655,432.052,172.025,27.046,154.995
C08773=1063.562,14.904,432.037,172.026,27.048,154.995
C08774=1063.568,15.153,432.022,172.027,27.051,154.995
C08775=1063.574,15.403,432.007,172.029,27.054,154.996
C08776=1063.580,15.652,431.992,172.030,27.056,154.996
C08777=1063.586,15.901,431.977,172.032,27.059,154.996
C08778=1063.592,16.151,431.961,172.033,27.061,154.997
C08779=1063.598,16.401,431.946,172.035,27.064,154.997
C08780=1063.604,16.650,431.932,172.036,27.066,154.997
C08781=1063.610,16.900,431.916,172.038,27.069,154.998
C08782=1063.616,17.149,431.901,172.040,27.071,154.998
C08783=1063.622,17.398,431.886,172.041,27.074,154.998
C08784=1063.628,17.648,431.870,172.043,27.076,154.999
C08785=1063.634,17.897,431.855,172.043,27.079,154.999
C08786=1063.641,18.147,431.840,172.045,27.081,154.999
C08787=1063.647,18.396,431.824,172.046,27.084,155.000
C08788=1063.653,18.645,431.810,172.048,27.086,155.000
C08789=1063.659,18.895,431.795,172.049,27.089,155.000
C08790=1063.665,19.145,431.779,172.051,27.091,155.001
C08791=1063.671,19.395,431.764,172.052,27.094,155.001
C08792=1063.677,19.643,431.749,172.054,27.097,155.001
C08793=1063.683,19.893,431.733,172.055,27.099,155.002
C08794=1063.689,20.143,431.718,172.057,27.102,155.002
C08795=1063.695,20.392,431.702,172.057,27.104,155.002
C08796=1063.701,20.642,431.687,172.059,27.107,155.003
C08797=1063.706,20.891,431.672,172.060,27.109,155.003
C08798=1063.713,21.141,431.657,172.062,27.112,155.003
C08799=1063.719,21.390,431.641,172.063,27.114,155.004
C08800=1063.725,21.640,431.626,172.065,27.117,155.004
C08801=1063.730,21.889,431.611,172.066,27.120,155.004
C08802=1063.737,22.138,431.595,172.068,27.122,155.005
C08803=1063.743,22.387,431.580,172.070,27.125,155.005
C08804=1063.749,22.637,431.564,172.071,27.128,155.005
C08805=1063.756,22.886,431.549,172.073,27.130,155.006
C08806=1063.761,23.136,431.534,172.073,27.132,155.006
C08807=1063.767,23.385,431.518,172.075,27.135,155.007
C08808=1063.773,23.635,431.502,172.076,27.138,155.007
C08809=1063.779,23.884,431.488,172.078,27.140,155.007
C08810=1063.785,24.134,431.471,172.079,27.143,155.007
C08811=1063.792,24.383,431.456,172.081,27.145,155.008
C08812=1063.797,24.632,431.440,172.082,27.148,155.008
C08813=1063.803,24.882,431.425,172.084,27.151,155.009
C08814=1063.809,25.132,431.410,172.085,27.153,155.009
C08815=1063.815,25.381,431.394,172.087,27.156,155.009
C08816=1063.821,25.631,431.379,172.087,27.158,155.010
C08817=1063.827,25.880,431.362,172.089,27.161,155.010
C08818=1063.834,26.130,431.348,172.090,27.163,155.010
C08819=1063.840,26.379,431.331,172.092,27.166,155.011
C08820=1063.845,26.628,431.317,172.093,27.169,155.011
C08821=1063.851,26.877,431.300,172.095,27.171,155.011
C08822=1063.858,27.127,431.285,172.096,27.174,155.012
C08823=1063.864,27.376,431.269,172.098,27.176,155.012
C08824=1063.870,27.626,431.254,172.099,27.179,155.012
C08825=1063.876,27.875,431.238,172.101,27.182,155.013
C08826=1063.882,28.125,431.222,172.102,27.184,155.013
C08827=1063.888,28.374,431.207,172.103,27.186,155.013
C08828=1063.894,28.624,431.191,172.105,27.189,155.014
C08829=1063.900,28.873,431.176,172.106,27.192,155.014
C08830=1063.906,29.123,431.160,172.108,27.194,155.014
C08831=1063.912,29.372,431.144,172.109,27.197,155.015
C08832=1063.918,29.621,431.128,172.111,27.199,155.015
C08833=1063.925,29.906,431.111,172.112,27.202,155.015
C08834=1063.932,30.190,431.093,172.114,27.206,155.016
C08835=1063.938,30.473,431.074,172.115,27.209,155.016
C08836=1063.945,30.758,431.057,172.116,27.211,155.017
C08837=1063.951,31.007,431.041,172.118,27.214,155.017
C08838=1063.957,31.256,431.025,172.120,27.217,155.017
C08839=1063.963,31.506,431.010,172.121,27.219,155.018
C08840=1063.969,31.755,430.993,172.123,27.222,155.018
C08841=1063.975,32.005,430.977,172.124,27.224,155.018
C08842=1063.981,32.254,430.962,172.126,27.227,155.019
C08843=1063.987,32.504,430.946,172.127,27.230,155.019
C08844=1063.993,32.753,430.930,172.129,27.232,155.020
C08845=1063.999,33.003,430.914,172.130,27.235,155.020
C08846=1064.006,33.252,430.898,172.131,27.237,155.020
C08847=1064.011,33.501,430.882,172.132,27.240,155.021
C08848=1064.017,33.751,430.867,172.134,27.243,155.021
C08849=1064.022,34.000,430.851,172.135,27.245,155.021
C08850=1064.029,34.249,430.835,172.137,27.248,155.022
C08851=1064.035,34.498,430.819,172.138,27.251,155.022
C08852=1064.041,34.748,430.803,172.140,27.253,155.022
C08853=1064.047,34.998,430.787,172.141,27.256,155.023
C08854=1064.053,35.247,430.771,172.143,27.259,155.023
C08855=1064.059,35.496,430.755,172.144,27.261,155.023
C08856=1064.065,35.746,430.740,172.145,27.264,155.024
C08857=1064.071,35.995,430.723,172.146,27.266,155.024
C08858=1064.077,36.245,430.707,172.148,27.269,155.025
C08859=1064.084,36.494,430.691,172.149,27.272,155.025
C08860=1064.090,36.743,430.675,172.151,27.274,155.025
C08861=1064.095,36.993,430.660,172.153,27.277,155.026
C08862=1064.101,37.243,430.643,172.154,27.280,155.026
C08863=1064.108,37.492,430.628,172.156,27.282,155.026
C08864=1064.114,37.741,430.611,172.157,27.285,155.027
C08865=1064.120,37.990,430.595,172.159,27.287,155.027
C08866=1064.126,38.240,430.579,172.159,27.289,155.027
C08867=1064.131,38.490,430.563,172.161,27.292,155.028
C08868=1064.137,38.739,430.547,172.162,27.295,155.028
C08869=1064.143,38.988,430.531,172.164,27.298,155.029
C08870=1064.149,39.238,430.515,172.165,27.300,155.029
C08871=1064.155,39.487,430.498,172.167,27.303,155.029
C08872=1064.161,39.736,430.482,172.168,27.306,155.030
C08873=1064.167,39.986,430.466,172.170,27.309,155.030
C08874=1064.173,40.235,430.450,172.171,27.311,155.030
C08875=1064.179,40.484,430.433,172.172,27.314,155.031
C08876=1064.185,40.734,430.417,172.173,27.316,155.031
C08877=1064.191,40.984,430.400,172.175,27.319,155.031
C08878=1064.197,41.233,430.384,172.176,27.321,155.032
C08879=1064.203,41.482,430.368,172.178,27.324,155.032
C08880=1064.209,41.732,430.352,172.179,27.327,155.033
C08881=1064.215,41.982,430.336,172.181,27.329,155.033
C08882=1064.221,42.231,430.320,172.182,27.332,155.033
C08883=1064.227,42.480,430.304,172.184,27.335,155.034
C08884=1064.233,42.730,430.287,172.184,27.338,155.034
C08885=1064.239,42.979,430.271,172.186,27.340,155.034
C08886=1064.245,43.229,430.255,172.188,27.343,155.035
C08887=1064.251,43.478,430.239,172.189,27.346,155.035
C08888=1064.257,43.727,430.222,172.191,27.348,155.035
C08889=1064.263,43.976,430.205,172.192,27.351,155.036
C08890=1064.269,44.225,430.189,172.194,27.353,155.036
C08891=1064.275,44.475,430.173,172.195,27.356,155.037
C08892=1064.280,44.724,430.156,172.197,27.359,155.037
C08893=1064.286,44.974,430.140,172.198,27.362,155.037
C08894=1064.292,45.223,430.123,172.199,27.364,155.038
C08895=1064.298,45.473,430.107,172.200,27.367,155.038
C08896=1064.304,45.723,430.090,172.202,27.370,155.038
C08897=1064.311,46.007,430.072,172.203,27.373,155.039
C08898=1064.318,46.290,430.053,172.205,27.376,155.039
C08899=1064.324,46.574,430.034,172.207,27.379,155.040
C08900=1064.331,46.859,430.015,172.208,27.382,155.040
C08901=1064.337,47.108,429.999,172.210,27.385,155.041
C08902=1064.342,47.357,429.982,172.212,27.387,155.041
C08903=1064.348,47.606,429.965,172.212,27.390,155.041
C08904=1064.354,47.856,429.949,172.214,27.393,155.042
C08905=1064.360,48.105,429.933,172.215,27.396,155.042
C08906=1064.365,48.355,429.916,172.217,27.398,155.043
C08907=1064.372,48.603,429.899,172.218,27.401,155.043
C08908=1064.377,48.853,429.883,172.220,27.403,155.043
C08909=1064.384,49.103,429.866,172.221,27.406,155.044
C08910=1064.389,49.352,429.849,172.223,27.409,155.044
C08911=1064.395,49.602,429.833,172.224,27.412,155.044
C08912=1064.401,49.850,429.816,172.225,27.414,155.045
C08913=1064.407,50.100,429.800,172.226,27.417,155.045
C08914=1064.413,50.349,429.783,172.228,27.420,155.045
C08915=1064.419,50.599,429.767,172.229,27.422,155.046
C08916=1064.425,50.848,429.749,172.231,27.425,155.046
C08917=1064.431,51.098,429.733,172.232,27.427,155.047
C08918=1064.437,51.347,429.716,172.234,27.430,155.047
C08919=1064.443,51.596,429.699,172.235,27.433,155.047
C08920=1064.449,51.845,429.683,172.237,27.436,155.048
C08921=1064.454,52.095,429.666,172.238,27.439,155.048
C08922=1064.461,52.345,429.649,172.239,27.441,155.048
C08923=1064.467,52.594,429.632,172.241,27.444,155.049
C08924=1064.473,52.843,429.616,172.242,27.446,155.049
C08925=1064.478,53.093,429.599,172.244,27.449,155.050
C08926=1064.484,53.342,429.582,172.245,27.452,155.050
C08927=1064.491,53.592,429.566,172.247,27.454,155.050
C08928=1064.496,53.841,429.549,172.248,27.457,155.051
C08929=1064.502,54.090,429.532,172.250,27.460,155.051
C08930=1064.508,54.339,429.516,172.251,27.463,155.051
C08931=1064.514,54.588,429.498,172.252,27.465,155.052
C08932=1064.520,54.838,429.482,172.253,27.468,155.052
C08933=1064.526,55.088,429.465,172.255,27.470,155.053
C08934=1064.532,55.336,429.448,172.256,27.473,155.053
C08935=1064.538,55.586,429.431,172.258,27.476,155.053
C08936=1064.545,55.836,429.414,172.259,27.478,155.054
C08937=1064.550,56.085,429.398,172.261,27.481,155.054
C08938=1064.556,56.335,429.381,172.262,27.484,155.054
C08939=1064.562,56.583,429.364,172.264,27.487,155.055
C08940=1064.569,56.833,429.347,172.265,27.490,155.055
C08941=1064.574,57.082,429.330,172.266,27.492,155.056
C08942=1064.580,57.332,429.314,172.268,27.494,155.056
C08943=1064.586,57.580,429.297,172.269,27.497,155.056
C08944=1064.592,57.831,429.279,172.271,27.500,155.057
C08945=1064.598,58.080,429.262,172.272,27.502,155.057
C08946=1064.604,58.329,429.246,172.274,27.505,155.057
C08947=1064.610,58.579,429.228,172.275,27.508,155.058
C08948=1064.616,58.828,429.212,172.277,27.511,155.058
C08949=1064.623,59.077,429.195,172.278,27.513,155.058
C08950=1064.628,59.327,429.178,172.280,27.516,155.059
C08951=1064.635,59.576,429.161,172.280,27.518,155.059
C08952=1064.640,59.825,429.144,172.282,27.521,155.060
C08953=1064.646,60.074,429.127,172.283,27.523,155.060
C08954=1064.653,60.324,429.110,172.285,27.526,155.060
C08955=1064.658,60.573,429.093,172.286,27.529,155.061
C08956=1064.665,60.823,429.075,172.288,27.532,155.061
C08957=1064.671,61.072,429.059,172.290,27.534,155.061
C08958=1064.677,61.321,429.042,172.291,27.537,155.062
C08959=1064.683,61.571,429.024,172.293,27.540,155.062
C08960=1064.689,61.820,429.007,172.294,27.543,155.063
C08961=1064.695,62.104,428.988,172.296,27.545,155.063
C08962=1064.702,62.387,428.969,172.297,27.548,155.063
C08963=1064.710,62.672,428.949,172.299,27.551,155.064
C08964=1064.716,62.955,428.930,172.300,27.554,155.064
C08965=1064.723,63.204,428.913,172.302,27.557,155.065
C08966=1064.729,63.454,428.896,172.303,27.559,155.065
C08967=1064.735,63.703,428.879,172.305,27.562,155.065
C08968=1064.741,63.952,428.862,172.306,27.564,155.066
C08969=1064.747,64.202,428.844,172.308,27.567,155.066
C08970=1064.753,64.451,428.827,172.309,27.570,155.066
C08971=1064.759,64.701,428.809,172.311,27.573,155.067
C08972=1064.765,64.949,428.793,172.312,27.576,155.067
C08973=1064.771,65.199,428.776,172.313,27.578,155.068
C08974=1064.777,65.449,428.758,172.314,27.581,155.068
C08975=1064.783,65.697,428.741,172.316,27.583,155.068
C08976=1064.788,65.947,428.724,172.317,27.586,155.069
C08977=1064.795,66.197,428.707,172.319,27.589,155.069
C08978=1064.801,66.446,428.689,172.320,27.592,155.070
C08979=1064.806,66.695,428.671,172.322,27.594,155.070
C08980=1064.813,66.944,428.654,172.324,27.597,155.070
C08981=1064.818,67.194,428.637,172.325,27.600,155.071
C08982=1064.824,67.443,428.619,172.327,27.602,155.071
C08983=1064.831,67.692,428.602,172.328,27.605,155.071
C08984=1064.836,67.941,428.585,172.329,27.608,155.072
C08985=1064.842,68.191,428.567,172.330,27.610,155.072
C08986=1064.848,68.440,428.551,172.332,27.613,155.073
C08987=1064.854,68.690,428.533,172.333,27.616,155.073
C08988=1064.860,68.939,428.515,172.335,27.618,155.073
C08989=1064.866,69.188,428.498,172.336,27.621,155.074
C08990=1064.872,69.438,428.480,172.338,27.624,155.074
C08991=1064.878,69.687,428.463,172.340,27.626,155.074
C08992=1064.885,69.936,428.445,172.341,27.629,155.075
C08993=1064.890,70.185,428.428,172.343,27.632,155.075
C08994=1064.896,70.435,428.410,172.344,27.635,155.076
C08995=1064.901,70.684,428.393,172.345,27.637,155.076
C08996=1064.907,70.933,428.375,172.346,27.640,155.076
C08997=1064.914,71.183,428.358,172.348,27.643,155.077
C08998=1064.919,71.432,428.340,172.349,27.646,155.077
C08999=1064.925,71.682,428.323,172.351,27.648,155.077
C09000=1064.931,71.931,428.305,172.352,27.651,155.078
C09001=1064.937,72.180,428.287,172.354,27.654,155.078
C09002=1064.943,72.429,428.270,172.355,27.656,155.079
C09003=1064.949,72.678,428.252,172.357,27.659,155.079
C09004=1064.955,72.928,428.235,172.358,27.662,155.079
C09005=1064.961,73.177,428.217,172.360,27.665,155.080
C09006=1064.967,73.427,428.199,172.360,27.667,155.080
C09007=1064.972,73.676,428.181,172.362,27.670,155.081
C09008=1064.979,73.925,428.164,172.364,27.672,155.081
C09009=1064.985,74.174,428.147,172.365,27.675,155.081
C09010=1064.991,74.424,428.129,172.367,27.678,155.082
C09011=1064.996,74.673,428.111,172.368,27.681,155.082
C09012=1065.002,74.923,428.093,172.370,27.684,155.083
C09013=1065.008,75.172,428.076,172.371,27.686,155.083
C09014=1065.014,75.422,428.058,172.373,27.689,155.083
C09015=1065.020,75.670,428.041,172.374,27.691,155.084
C09016=1065.026,75.920,428.023,172.376,27.694,155.084
C09017=1065.032,76.168,428.004,172.377,27.697,155.084
C09018=1065.038,76.418,427.987,172.378,27.700,155.085
C09019=1065.044,76.667,427.969,172.379,27.702,155.085
C09020=1065.050,76.917,427.951,172.381,27.705,155.086
C09021=1065.055,77.166,427.933,172.383,27.707,155.086
C09022=1065.062,77.416,427.916,172.384,27.710,155.086
C09023=1065.067,77.665,427.898,172.386,27.713,155.087
C09024=1065.074,77.914,427.881,172.387,27.716,155.087
C09025=1065.080,78.198,427.860,172.389,27.719,155.088
C09026=1065.087,78.481,427.839,172.390,27.722,155.088
C09027=1065.094,78.765,427.820,172.393,27.725,155.088
C09028=1065.100,79.048,427.799,172.394,27.728,155.089
C09029=1065.107,79.298,427.781,172.396,27.731,155.089
C09030=1065.112,79.547,427.763,172.397,27.733,155.090
C09031=1065.119,79.796,427.745,172.398,27.736,155.090
C09032=1065.123,80.046,427.727,172.399,27.739,155.090
C09033=1065.129,80.295,427.709,172.401,27.742,155.091
C09034=1065.135,80.544,427.691,172.402,27.744,155.091
C09035=1065.141,80.793,427.672,172.404,27.747,155.092
C09036=1065.147,81.042,427.655,172.405,27.750,155.092
C09037=1065.153,81.292,427.637,172.407,27.753,155.092
C09038=1065.159,81.541,427.619,172.408,27.756,155.093
C09039=1065.165,81.790,427.601,172.410,27.758,155.093
C09040=1065.170,82.039,427.583,172.412,27.761,155.094
C09041=1065.177,82.289,427.565,172.413,27.764,155.094
C09042=1065.182,82.538,427.546,172.415,27.767,155.094
C09043=1065.188,82.788,427.528,172.416,27.770,155.095
C09044=1065.194,83.037,427.511,172.417,27.772,155.095
C09045=1065.200,83.286,427.492,172.418,27.774,155.096
C09046=1065.206,83.536,427.474,172.420,27.777,155.096
C09047=1065.211,83.785,427.457,172.421,27.780,155.096
C09048=1065.218,84.034,427.438,172.423,27.783,155.097
C09049=1065.224,84.283,427.420,172.424,27.786,155.097
C09050=1065.229,84.533,427.402,172.426,27.788,155.098
C09051=1065.235,84.782,427.383,172.427,27.791,155.098
C09052=1065.241,85.031,427.366,172.429,27.794,155.098
C09053=1065.247,85.280,427.347,172.431,27.796,155.099
C09054=1065.253,85.530,427.329,172.432,27.799,155.099
C09055=1065.259,85.779,427.312,172.434,27.802,155.099
C09056=1065.265,86.028,427.293,172.435,27.805,155.100
C09057=1065.270,86.277,427.275,172.437,27.807,155.100
C09058=1065.276,86.526,427.256,172.438,27.810,155.101
C09059=1065.282,86.776,427.238,172.439,27.813,155.101
C09060=1065.288,87.025,427.220,172.440,27.815,155.101
C09061=1065.294,87.274,427.202,172.442,27.818,155.102
C09062=1065.301,87.524,427.184,172.444,27.820,155.102
C09063=1065.306,87.773,427.165,172.445,27.823,155.103
C09064=1065.312,88.023,427.147,172.447,27.826,155.103
C09065=1065.318,88.272,427.129,172.448,27.829,155.103
C09066=1065.324,88.521,427.111,172.450,27.832,155.104
C09067=1065.330,88.770,427.092,172.451,27.834,155.104
C09068=1065.336,89.020,427.074,172.453,27.837,155.104
C09069=1065.341,89.268,427.056,172.454,27.839,155.105
C09070=1065.348,89.517,427.037,172.456,27.842,155.105
C09071=1065.354,89.767,427.019,172.457,27.845,155.106
C09072=1065.360,90.016,427.000,172.459,27.848,155.106
C09073=1065.366,90.265,426.983,172.461,27.851,155.106
C09074=1065.372,90.515,426.964,172.462,27.853,155.107
C09075=1065.378,90.765,426.946,172.464,27.856,155.107
C09076=1065.383,91.013,426.927,172.465,27.858,155.108
C09077=1065.389,91.262,426.908,172.466,27.861,155.108
C09078=1065.395,91.512,426.890,172.467,27.864,155.108
C09079=1065.401,91.761,426.872,172.469,27.867,155.109
C09080=1065.406,92.011,426.853,172.470,27.869,155.109
C09081=1065.413,92.260,426.835,172.472,27.872,155.110
C09082=1065.418,92.508,426.816,172.474,27.875,155.110
C09083=1065.424,92.758,426.798,172.475,27.878,155.110
C09084=1065.430,93.008,426.779,172.477,27.880,155.111
C09085=1065.436,93.257,426.760,172.478,27.883,155.111
C09086=1065.442,93.506,426.742,172.480,27.886,155.112
C09087=1065.447,93.755,426.723,172.481,27.889,155.112
C09088=1065.454,94.004,426.705,172.483,27.892,155.112
C09089=1065.460,94.288,426.684,172.484,27.894,155.113
C09090=1065.466,94.572,426.662,172.486,27.898,155.113
C09091=1065.473,94.855,426.642,172.488,27.901,155.114
C09092=1065.480,95.138,426.620,172.490,27.904,155.114
C09093=1065.486,95.389,426.601,172.491,27.906,155.114
C09094=1065.492,95.638,426.583,172.493,27.909,155.115
C09095=1065.498,95.886,426.564,172.494,27.912,155.115
C09096=1065.503,96.135,426.545,172.496,27.915,155.116
C09097=1065.510,96.385,426.527,172.497,27.918,155.116
C09098=1065.515,96.635,426.508,172.499,27.920,155.116
C09099=1065.521,96.883,426.490,172.501,27.923,155.117
C09100=1065.527,97.133,426.471,172.501,27.926,155.117
C09101=1065.533,97.382,426.452,172.503,27.928,155.118
C09102=1065.539,97.632,426.433,172.504,27.931,155.118
C09103=1065.545,97.881,426.415,172.506,27.933,155.118
C09104=1065.550,98.130,426.396,172.507,27.936,155.119
C09105=1065.557,98.379,426.377,172.509,27.939,155.119
C09106=1065.562,98.628,426.358,172.510,27.942,155.120
C09107=1065.569,98.877,426.339,172.512,27.945,155.120
